// TIA Portal project "Project1" (V14)

(* hardware
DEVICE "S71500/ET200MP station_1"  S7-1500 station
   slot 0: "Rail_0"  Rack  6ES7 590-1***0-0AA0
   slot 1: "PLC_1"  CPU 1516-3 PN/DP  6ES7 516-3AN01-0AB0  V2.1
      slot 3: "CPU display_1"  6ES7591-1BA00-0AA0
   slot 2: "DI 16x24VDC SRC BA_1"  DI 16x24VDC SRC BA  6ES7 521-1BH50-0AA0  V2.0
   slot 3: "DI 16/DQ 16x24VDC/0.5A BA_1"  DI 16/DQ 16x24VDC/0.5A BA  6ES7 523-1BL00-0AA0  V1.0
   slot 4: "AI 8xU/R/RTD/TC HF_1"  AI 8xU/R/RTD/TC HF  6ES7 531-7PF00-0AB0  V1.1
   slot 5: "AQ 4xU/I HF_1"  AQ 4xU/I HF  6ES7 532-5ND00-0AB0  V1.1
   slot 6: "AI/AQ 4xU/I/RTD/TC / 2xU/I ST_1"  AI/AQ 4xU/I/RTD/TC / 2xU/I ST  6ES7 534-7QE00-0AB0  V1.0
   slot 7: "DQ 16x24VDC/0.5A BA_1"  DQ 16x24VDC/0.5A BA  6ES7 522-1BH10-0AA0  V1.0
*)

// ===== PLC "PLC_1"  CPU 1516-3 PN/DP =====

VAR_GLOBAL   // PLC tag table "UP_Robot1"
   "robot1_dc" AT %E0.7 : Bool;
   "robot1_fin_p" AT %E1.0 : Bool;
   "robot1_home" AT %E1.1 : Bool;
   "robot1_temp" AT %T1 : Timer;
   "robot1_cargar" AT %A1.2 : Bool;
   "robot1_descargar" AT %A1.3 : Bool;
   "robot1_b_standby" AT %M1.4 : Bool;   // b = bit
   "robot1_b_ocupacion" AT %M1.5 : Bool;
   "robot1_bdt_carga" AT %M1.6 : Bool;   // bdt = bit de tiempo
   "robot1_bdt_descarga" AT %M1.7 : Bool;
   "robot1_bdc_carga" AT %M2.0 : Bool;   // bdc = bit de configuración
   "robot1_bdc_descarga" AT %M2.1 : Bool;
   "robot1_b_emer" AT %M2.2 : Bool;
   "robot1_emer" AT %M5.7 : Bool;
   "robot1_rearme" AT %M6.0 : Bool;
   "robot1_x_emer" AT %M5.5 : Bool;
   "robot1_x_marcha" AT %M5.6 : Bool;
END_VAR

VAR_GLOBAL   // PLC tag table "UP_Robot2"
   "robot2_dc" AT %E2.5 : Bool;
   "robot2_fin_p" AT %E2.6 : Bool;
   "robot2_home" AT %E3.6 : Bool;
   "robot2_temp" AT %T5 : Timer;
   "robot2_cargar" AT %A6.0 : Bool;
   "robot2_descargar" AT %A6.1 : Bool;
   "robot2_b_standby" AT %M6.2 : Bool;   // b = bit
   "robot2_b_ocupacion" AT %M6.3 : Bool;
   "robot2_bdt_carga" AT %M6.4 : Bool;   // bdt = bit de tiempo
   "robot2_bdt_descarga" AT %M6.5 : Bool;
   "robot2_bdc_carga" AT %M6.6 : Bool;   // bdc = bit de configuración
   "robot2_bdc_descarga" AT %M6.7 : Bool;
   "robot2_b_emer" AT %M7.0 : Bool;
   "robot2_emer" AT %E4.6 : Bool;
   "robot2_rearme" AT %E4.7 : Bool;
END_VAR

VAR_GLOBAL   // PLC tag table "GMM"
   "gmm_on" AT %E0.0 : Bool;
   "gmm_lote_pequenio" AT %E0.1 : Bool;
   "gmm_lote_mediano" AT %E0.2 : Bool;
   "gmm_lote_grande" AT %E0.3 : Bool;
   "gmm_mcong" AT %E0.4 : Bool;
   "gmm_cong" AT %E0.5 : Bool;
   "gmm_bit_marcha" AT %M0.6 : Bool;
   "gmm_bit_paro" AT %M0.7 : Bool;
   "gmm_bit_congelacion" AT %M1.0 : Bool;
END_VAR

VAR_GLOBAL   // PLC tag table "CeldaMecanizado"
   "start" AT %E0.6 : Bool;
END_VAR

VAR_GLOBAL   // PLC tag table "UP_CNC1"
   "cnc1_lapiz" AT %E1.2 : Bool;
   "cnc1_sacapuntas" AT %E1.3 : Bool;
   "cnc1_escuadra" AT %E1.4 : Bool;
   "cnc1_cartabon" AT %E1.5 : Bool;
   "cnc1_home" AT %E1.6 : Bool;
   "cnc1_temp" AT %T2 : Timer;
   "cnc1_cnc_lapiz" AT %A1.7 : Bool;
   "cnc1_cnc_sacapuntas" AT %A2.0 : Bool;
   "cnc1_cnc_escuadra" AT %A2.1 : Bool;
   "cnc1_cnc_cartabon" AT %A2.2 : Bool;
   "cnc1_b_standby" AT %M2.3 : Bool;   // b = bit
   "cnc1_b_ocupacion" AT %M2.4 : Bool;
   "cnc1_bdt_lapiz" AT %M2.5 : Bool;   // bdt = bit de tiempo
   "cnc1_bdt_sacapuntas" AT %M2.6 : Bool;
   "cnc1_bdt_escuadra" AT %M2.7 : Bool;
   "cnc1_bdt_cartabon" AT %M3.0 : Bool;
   "cnc1_bdc_lapiz" AT %M3.1 : Bool;   // bdc = bit de configuración
   "cnc1_bdc_sacapuntas" AT %M3.2 : Bool;
   "cnc1_bdc_escuadra" AT %M3.3 : Bool;
   "cnc1_bdc_cartabon" AT %M3.4 : Bool;
   "cnc1_b_emer" AT %M3.5 : Bool;
   "cnc1_emer" AT %M6.1 : Bool;
   "cnc1_rearme" AT %M7.3 : Bool;
END_VAR

VAR_GLOBAL   // PLC tag table "UP_Simple_Efecto1"
   "sef1_scomp" AT %E1.7 : Bool;   // sef = simple efecto
   "sef1_sexp" AT %E2.0 : Bool;
   "sef1_push" AT %E2.1 : Bool;
   "sef1_temp" AT %T3 : Timer;
   "sef1_expandir" AT %A2.3 : Bool;
   "sef1_b_standby" AT %M3.6 : Bool;   // b = bit
   "sef1_b_ocupacion" AT %M3.7 : Bool;
   "sef1_bdt_expansion" AT %M4.0 : Bool;   // bdt = bit de tiempo
   "sef1_bdt_compresion" AT %M4.1 : Bool;
   "sef1_bdc_expansion" AT %M4.2 : Bool;   // bdc = bit de configuración
   "sef1_bdc_compresion" AT %M4.3 : Bool;
   "sef1_b_emer" AT %M4.4 : Bool;
   "sef1_emer" AT %M9.1 : Bool;
   "sef1_rearme" AT %M9.2 : Bool;
END_VAR

VAR_GLOBAL   // PLC tag table "UT"
   "ut_x0" AT %M4.5 : Bool;
   "ut_m1" AT %M4.6 : Bool;
   "ut_x2" AT %M4.7 : Bool;
   "ut_x10" AT %M5.0 : Bool;
   "ut_r1" AT %E2.2 : Bool;
   "ut_r2" AT %E2.3 : Bool;
   "ut_rearme" AT %E2.4 : Bool;
   "ut_emer" AT %E2.7 : Bool;
   "ut_cong" AT %E3.0 : Bool;
   "ut_sini" AT %E3.1 : Bool;
   "ut_sfin" AT %E3.2 : Bool;
   "ut_reset" AT %E3.3 : Bool;
   "ut_bdt" AT %M5.1 : Bool;   // bdt = bit de tiempo
   "ut_bdc" AT %M5.2 : Bool;   // bdc = bit de configuración
   "ut_bdf" AT %M5.3 : Bool;   // bdf = bit de fin
   "ut_bdo" AT %M5.4 : Bool;   // bdo = bit de ocupación
   "ut_s1" AT %E3.4 : Bool;
   "ut_s2" AT %E3.5 : Bool;
   "ut_temp" AT %T4 : Timer;
   "ut_actuador1" AT %A3.6 : Bool;
END_VAR

VAR_GLOBAL   // PLC tag table "UP_CNC2"
   "cnc2_lapiz" AT %E3.7 : Bool;
   "cnc2_sacapuntas" AT %E4.0 : Bool;
   "cnc2_escuadra" AT %E4.1 : Bool;
   "cnc2_cartabon" AT %E4.2 : Bool;
   "cnc2_home" AT %E4.3 : Bool;
   "cnc2_temp" AT %T6 : Timer;
   "cnc2_cnc_lapiz" AT %A7.0 : Bool;
   "cnc2_cnc_sacapuntas" AT %A7.1 : Bool;
   "cnc2_cnc_escuadra" AT %A7.2 : Bool;
   "cnc2_cnc_cartabon" AT %A7.3 : Bool;
   "cnc2_b_standby" AT %M7.4 : Bool;   // b = bit
   "cnc2_b_ocupacion" AT %M7.5 : Bool;
   "cnc2_bdt_lapiz" AT %M7.6 : Bool;   // bdt = bit de tiempo
   "cnc2_bdt_sacapuntas" AT %M7.7 : Bool;
   "cnc2_bdt_escuadra" AT %M8.0 : Bool;
   "cnc2_bdt_cartabon" AT %M8.1 : Bool;
   "cnc2_bdc_lapiz" AT %M8.2 : Bool;   // bdc = bit de configuración
   "cnc2_bdc_sacapuntas" AT %M8.3 : Bool;
   "cnc2_bdc_escuadra" AT %M8.4 : Bool;
   "cnc2_bdc_cartabon" AT %M8.5 : Bool;
   "cnc2_b_emer" AT %M8.6 : Bool;
   "cnc2_emer" AT %M8.7 : Bool;
   "cnc2_rearme" AT %M9.0 : Bool;
END_VAR

VAR_GLOBAL   // PLC tag table "GEMER"
   "x_emer" AT %M7.1 : Bool;
   "x_marcha" AT %M7.2 : Bool;
   "emer" AT %E5.0 : Bool;
   "rearme" AT %E5.1 : Bool;
   "emer_local_robot1" AT %E5.2 : Bool;
   "rearme_local_robot1" AT %E5.3 : Bool;
   "emer_local_robot2" AT %E5.4 : Bool;
   "rearme_local_robot2" AT %E5.5 : Bool;
   "emer_local_cnc1" AT %E5.6 : Bool;
   "rearme_local_cnc1" AT %E5.7 : Bool;
   "emer_local_simple_efecto1" AT %E6.0 : Bool;
   "rearme_local_simple_efecto1" AT %E6.1 : Bool;
   "emer_local_cnc2" AT %E6.2 : Bool;
   "rearme_local_cnc2" AT %E6.3 : Bool;
   "emer_local_palets_vacios" AT %E6.4 : Bool;
   "rearme_local_palets_vacios" AT %E6.5 : Bool;
END_VAR

VAR_GLOBAL   // PLC tag table "UP_Palets_Vacios"
   "pa_emer" AT %M9.3 : Bool;
   "pa_rearme" AT %M9.4 : Bool;
   "pa_recoger_pila" AT %A9.5 : Bool;
   "pa_pila_saturada" AT %A9.6 : Bool;
   "pa_error_medida" AT %A9.7 : Bool;
   "pa_h<hmin" AT %A10.0 : Bool;
   "pa_h>hmin" AT %A10.1 : Bool;
   "pa_h>hmax" AT %A10.2 : Bool;
   "pa_hreal" AT %AD10 : Real;
   "pa_hraw" AT %EW14 : Int;
END_VAR

// folder: CNC

DATA_BLOCK "UP_CNC1_DB"   // DB4
{ S7_Optimized_Access := 'TRUE' }
VERSION : 0.1
// stored: InstanceOfName UP_CNC
"UP_CNC"
BEGIN
END_DATA_BLOCK

DATA_BLOCK "UP_CNC2_DB"   // DB18
{ S7_Optimized_Access := 'TRUE' }
VERSION : 0.1
// stored: InstanceOfName UP_CNC
"UP_CNC"
BEGIN
END_DATA_BLOCK

// folder: Cilindro simple efecto

DATA_BLOCK "UP_Simple_Efecto1_DB"   // DB10
{ S7_Optimized_Access := 'TRUE' }
VERSION : 0.1
// stored: InstanceOfName UP_Simple_Efecto
"UP_Simple_Efecto"
BEGIN
END_DATA_BLOCK

// folder: Datos producción

DATA_BLOCK "datosProduccion"   // DB1
{ S7_Optimized_Access := 'TRUE' }
VERSION : 0.1
   VAR
      tmax_simple_efecto : S5Time := s5t#5s;   // Tiempo máximo expansión / compresión
      tmax_carga_descarga : S5Time := s5t#10s;   // Tiempo máximo carga / descarga
      tmax_cnc_lapiz : S5Time := s5t#14s;   // Tiempo máximo cnc
      tmax_cnc_sacapuntas : S5Time := s5t#20s;
      tmax_cnc_escuadra : S5Time := s5t#10s;
      tmax_cnc_cartabon : S5Time := s5t#10s;
      LO_LIM : Real := 0.0;
      HI_LIM : Real := 50.0;
      hmin : Real := 25.0;
      hmax : Real := 30.0;
   END_VAR
BEGIN
END_DATA_BLOCK

DATA_BLOCK "datosLotePequenio"   // DB8
{ S7_Optimized_Access := 'TRUE' }
VERSION : 0.1
   VAR
      tmax_cnc_lapiz : S5Time := s5t#7s;   // Tiempo máximo cnc
      tmax_cnc_sacapuntas : S5Time := s5t#10s;
      tmax_cnc_escuadra : S5Time := s5t#5s;
      tmax_cnc_cartabon : S5Time := s5t#5s;
   END_VAR
BEGIN
END_DATA_BLOCK

DATA_BLOCK "datosLoteMediano"   // DB9
{ S7_Optimized_Access := 'TRUE' }
VERSION : 0.1
   VAR
      tmax_cnc_lapiz : S5Time := s5t#14s;   // Tiempo máximo cnc
      tmax_cnc_sacapuntas : S5Time := s5t#20s;
      tmax_cnc_escuadra : S5Time := s5t#10s;
      tmax_cnc_cartabon : S5Time := s5t#10s;
   END_VAR
BEGIN
END_DATA_BLOCK

DATA_BLOCK "datosLoteGrande"   // DB12
{ S7_Optimized_Access := 'TRUE' }
VERSION : 0.1
   VAR
      tmax_cnc_lapiz : S5Time := s5t#21s;   // Tiempo máximo cnc
      tmax_cnc_sacapuntas : S5Time := s5t#30s;
      tmax_cnc_escuadra : S5Time := s5t#15s;
      tmax_cnc_cartabon : S5Time := s5t#15s;
   END_VAR
BEGIN
END_DATA_BLOCK

// folder: Emergencia

DATA_BLOCK "GEMER_Robot1_DB"   // DB5
{ S7_Optimized_Access := 'TRUE' }
VERSION : 0.1
// stored: InstanceOfName GEMER_Local
"GEMER_Local"
BEGIN
END_DATA_BLOCK

DATA_BLOCK "GEMER_Robot2_DB"   // DB6
{ S7_Optimized_Access := 'TRUE' }
VERSION : 0.1
// stored: InstanceOfName GEMER_Local
"GEMER_Local"
BEGIN
END_DATA_BLOCK

DATA_BLOCK "GEMER_CNC1_DB"   // DB19
{ S7_Optimized_Access := 'TRUE' }
VERSION : 0.1
// stored: InstanceOfName GEMER_Local
"GEMER_Local"
BEGIN
END_DATA_BLOCK

DATA_BLOCK "GEMER_CNC2_DB"   // DB20
{ S7_Optimized_Access := 'TRUE' }
VERSION : 0.1
// stored: InstanceOfName GEMER_Local
"GEMER_Local"
BEGIN
END_DATA_BLOCK

DATA_BLOCK "GEMER_Simple_Efecto1_DB"   // DB21
{ S7_Optimized_Access := 'TRUE' }
VERSION : 0.1
// stored: InstanceOfName GEMER_Local
"GEMER_Local"
BEGIN
END_DATA_BLOCK

DATA_BLOCK "GEMER_Local_Palets_Vacios_DB"   // DB22
{ S7_Optimized_Access := 'TRUE' }
VERSION : 0.1
// stored: InstanceOfName GEMER_Local
"GEMER_Local"
BEGIN
END_DATA_BLOCK

// folder: Modos de marcha

DATA_BLOCK "GMM_DB"   // DB2
{ S7_Optimized_Access := 'TRUE' }
VERSION : 0.1
// stored: InstanceOfName GMM
"GMM"
BEGIN
END_DATA_BLOCK

// folder: Palets vacíos

DATA_BLOCK "UP_Palets_Vacios_DB"   // DB7
{ S7_Optimized_Access := 'TRUE' }
VERSION : 0.1
// stored: InstanceOfName UP_Palets_Vacios
"UP_Palets_Vacios"
BEGIN
END_DATA_BLOCK

// folder: Robots carga / descarga

DATA_BLOCK "UP_Robot1_DB"   // DB3
{ S7_Optimized_Access := 'TRUE' }
VERSION : 0.1
// stored: InstanceOfName UP_Robot
"UP_Robot"
BEGIN
END_DATA_BLOCK

DATA_BLOCK "UP_Robot2_DB"   // DB17
{ S7_Optimized_Access := 'TRUE' }
VERSION : 0.1
// stored: InstanceOfName UP_Robot
"UP_Robot"
BEGIN
END_DATA_BLOCK

// folder: Test unitarios

DATA_BLOCK "UT_SFC_Cilindro_DB"   // DB11
{ S7_Optimized_Access := 'TRUE' }
VERSION : 0.1
// stored: InstanceOfName SFC_Cilindro
"SFC_Cilindro"
BEGIN
END_DATA_BLOCK

DATA_BLOCK "UT_SFC_Programa_DB"   // DB13
{ S7_Optimized_Access := 'TRUE' }
VERSION : 0.1
// stored: InstanceOfName SFC_Programa
"SFC_Programa"
BEGIN
END_DATA_BLOCK

DATA_BLOCK "UT_UP_Simple_Efecto_DB"   // DB14
{ S7_Optimized_Access := 'TRUE' }
VERSION : 0.1
// stored: InstanceOfName UP_Simple_Efecto
"UP_Simple_Efecto"
BEGIN
END_DATA_BLOCK

DATA_BLOCK "UT_UP_CNC_DB"   // DB15
{ S7_Optimized_Access := 'TRUE' }
VERSION : 0.1
// stored: InstanceOfName UP_CNC
"UP_CNC"
BEGIN
END_DATA_BLOCK

DATA_BLOCK "UT_UP_Robot_DB"   // DB16
{ S7_Optimized_Access := 'TRUE' }
VERSION : 0.1
// stored: InstanceOfName UP_Robot
"UP_Robot"
BEGIN
END_DATA_BLOCK

DATA_BLOCK "UT_UP_Palets_Vacios_DB"   // DB23
{ S7_Optimized_Access := 'TRUE' }
VERSION : 0.1
// stored: InstanceOfName UP_Palets_Vacios
"UP_Palets_Vacios"
BEGIN
END_DATA_BLOCK

// folder: (top level)

ORGANIZATION_BLOCK "main"   // OB1, STL, ProgramCycle
TITLE = "Main Program Sweep (Cycle)"
{ S7_Optimized_Access := 'TRUE' }
VERSION : 0.1
// Se encarga de llamar a las unidades productivas, integrando los modos de marcha y las emergencias. Llama a los bloques en el siguiente orden:
// - Emergencia global
// - Emergencias locales
// - Rearmes
// - Modos de marcha
// - Unidades productivas
// Las salidas de los bloques de emergencia y modos de marcha determinarán las entradas “emer”, “rearme”, “cong” y “start” de las unidades productivas.
   VAR_INPUT
      Initial_Call : Bool;   // Initial call of this OB
      Remanence : Bool;   // =True, if remanent data are available
   END_VAR
BEGIN

REGION Network 1: Gemer global
   // Llama a la emergencia global.
         CALL  "GEMER_Global";
END_REGION

REGION Network 2: Gemer robot1
   // Si no hay emergencia global, llama a la emergencia del robot 1.
         AN    "x_emer";

         JCN   _emer_robot1;

         CALL  "GEMER_Local", "GEMER_Robot1_DB"
         ( emer     := "emer_local_robot1",
           rearme   := "rearme_local_robot1",
           bit_emer := "robot1_emer"
         );

   _emer_robot1:NOP   0;
END_REGION

REGION Network 3: Gemer robot2
   // Si no hay emergencia global, llama a la emergencia del robot 2.
         AN    "x_emer";

         JCN   _emer_robot2;

         CALL  "GEMER_Local", "GEMER_Robot2_DB"
         ( emer     := "emer_local_robot2",
           rearme   := "rearme_local_robot2",
           bit_emer := "robot2_emer"
         );

   _emer_robot2:NOP   0;
END_REGION

REGION Network 4: Gemer cnc1
   // Si no hay emergencia global, llama a la emergencia del cnc 1.
         AN    "x_emer";

         JCN   _emer_cnc1;

         CALL  "GEMER_Local", "GEMER_CNC1_DB"
         ( emer     := "emer_local_cnc1",
           rearme   := "rearme_local_cnc1",
           bit_emer := "cnc1_emer"
         );

   _emer_cnc1:NOP   0;
END_REGION

REGION Network 5: Gemer cnc2
   // Si no hay emergencia global, llama a la emergencia del cnc 2.
         AN    "x_emer";

         JCN   _emer_cnc2;

         CALL  "GEMER_Local", "GEMER_CNC2_DB"
         ( emer     := "emer_local_cnc2",
           rearme   := "rearme_local_cnc2",
           bit_emer := "cnc2_emer"
         );

   _emer_cnc2:NOP   0;
END_REGION

REGION Network 6: Gemer simple efecto1
         AN    "x_emer";

         JCN   _emer_simple_efecto1;

         CALL  "GEMER_Local", "GEMER_Simple_Efecto1_DB"
         ( emer     := "emer_local_simple_efecto1",
           rearme   := "rearme_local_simple_efecto1",
           bit_emer := "sef1_emer"
         );

   _emer_simple_efecto1:NOP   0;
END_REGION

REGION Network 7: Gemer palets vacíos
         AN    "x_emer";

         JCN   _palets_vacios1;

         CALL  "GEMER_Local", "GEMER_Local_Palets_Vacios_DB"
         ( emer     := "emer_local_palets_vacios",
           rearme   := "rearme_local_palets_vacios",
           bit_emer := "pa_emer"
         );

   _palets_vacios1:NOP   0;
END_REGION

REGION Network 8: Rearme robot1
         O     "rearme";
         O     "rearme_local_robot1";
         =     "robot1_rearme";
END_REGION

REGION Network 9: Rearme robot2
         O     "rearme";
         O     "rearme_local_robot2";
         =     "robot2_rearme";
END_REGION

REGION Network 10: Rearme cnc1
         O     "rearme";
         O     "rearme_local_cnc1";
         =     "cnc1_rearme";
END_REGION

REGION Network 11: Rearme cnc2
         O     "rearme";
         O     "rearme_local_cnc2";
         =     "cnc2_rearme";
END_REGION

REGION Network 12: Rearme simple efecto1
         O     "rearme";
         O     "rearme_local_simple_efecto1";
         =     "sef1_rearme";
END_REGION

REGION Network 13: Rearme palets vacíos
         O     "rearme";
         O     "rearme_local_palets_vacios";
         =     "pa_rearme";
END_REGION

REGION Network 14: GMM
   // Si no hay emergencia global, se ejecutan los modos de marcha. En caso contrario, se ejecutarán desde GEMER_Global, que activará la plantilla de desconexión:
         AN    "x_emer";

         JCN   _gmm_emer;

         CALL  "GMM", "GMM_DB"
         ( on              := "gmm_on",
           lote_pequenio   := "gmm_lote_pequenio",
           lote_mediano    := "gmm_lote_mediano",
           lote_grande     := "gmm_lote_grande",
           mcong           := "gmm_mcong",
           cong            := "gmm_cong",
           emer            := FALSE,
           bit_paro        := "gmm_bit_paro",
           bit_marcha      := "gmm_bit_marcha",
           bit_congelacion := "gmm_bit_congelacion"
         );

   _gmm_emer:NOP   0;
END_REGION

REGION Network 15: UP_Robot1
         CALL  "UP_Robot", "UP_Robot1_DB"
         ( start                     := "gmm_bit_marcha",
           emer                      := "robot1_emer",
           rearme                    := "robot1_rearme",
           cong                      := "gmm_bit_congelacion",
           dc                        := "robot1_dc",
           fin_p                     := "robot1_fin_p",
           home                      := "robot1_home",
           tiempo_max                := "datosProduccion".tmax_carga_descarga,
           temp_max                  := "robot1_temp",
           cargar                    := "robot1_cargar",
           descargar                 := "robot1_descargar",
           bit_standby               := "robot1_b_standby",
           bit_ocupacion             := "robot1_b_ocupacion",
           bit_error_tiempo_carga    := "robot1_bdt_carga",
           bit_error_tiempo_descarga := "robot1_bdt_descarga",
           bit_error_config_carga    := "robot1_bdc_carga",
           bit_error_config_descarga := "robot1_bdc_descarga",
           bit_emer                  := "robot1_b_emer"
         );
END_REGION

REGION Network 16: UP_Robot2
         CALL  "UP_Robot", "UP_Robot2_DB"
         ( start                     := "gmm_bit_marcha",
           emer                      := "robot2_emer",
           rearme                    := "robot2_rearme",
           cong                      := "gmm_bit_congelacion",
           dc                        := "robot2_dc",
           fin_p                     := "robot2_fin_p",
           home                      := "robot2_home",
           tiempo_max                := "datosProduccion".tmax_carga_descarga,
           temp_max                  := "robot2_temp",
           cargar                    := "robot2_cargar",
           descargar                 := "robot2_descargar",
           bit_standby               := "robot2_b_standby",
           bit_ocupacion             := "robot2_b_ocupacion",
           bit_error_tiempo_carga    := "robot2_bdt_carga",
           bit_error_tiempo_descarga := "robot2_bdt_descarga",
           bit_error_config_carga    := "robot2_bdc_carga",
           bit_error_config_descarga := "robot2_bdc_descarga",
           bit_emer                  := "robot2_b_emer"
         );
END_REGION

REGION Network 17: UP_CNC1
         CALL  "UP_CNC", "UP_CNC1_DB"
         ( start                       := "gmm_bit_marcha",
           emer                        := "cnc1_emer",
           rearme                      := "cnc1_rearme",
           cong                        := "gmm_bit_congelacion",
           lapiz                       := "cnc1_lapiz",
           sacapuntas                  := "cnc1_sacapuntas",
           escuadra                    := "cnc1_escuadra",
           cartabon                    := "cnc1_cartabon",
           home                        := "cnc1_home",
           tmax_cnc_lapiz              := "datosProduccion".tmax_cnc_lapiz,
           tmax_cnc_sacapuntas         := "datosProduccion".tmax_cnc_sacapuntas,
           tmax_cnc_escuadra           := "datosProduccion".tmax_cnc_escuadra,
           tmax_cnc_cartabon           := "datosProduccion".tmax_cnc_cartabon,
           temp_max                    := "cnc1_temp",
           cnc_lapiz                   := "cnc1_cnc_lapiz",
           cnc_sacapuntas              := "cnc1_cnc_sacapuntas",
           cnc_escuadra                := "cnc1_cnc_escuadra",
           cnc_cartabon                := "cnc1_cnc_cartabon",
           bit_standby                 := "cnc1_b_standby",
           bit_ocupacion               := "cnc1_b_ocupacion",
           bit_error_tiempo_lapiz      := "cnc1_bdt_lapiz",
           bit_error_tiempo_sacapuntas := "cnc1_bdt_sacapuntas",
           bit_error_tiempo_escuadra   := "cnc1_bdt_escuadra",
           bit_error_tiempo_cartabon   := "cnc1_bdt_cartabon",
           bit_error_config_lapiz      := "cnc1_bdc_lapiz",
           bit_error_config_sacapuntas := "cnc1_bdc_sacapuntas",
           bit_error_config_escuadra   := "cnc1_bdc_escuadra",
           bit_error_config_cartabon   := "cnc1_bdc_cartabon",
           bit_emer                    := "cnc1_b_emer"
         );
END_REGION

REGION Network 18: UP_CNC2
         CALL  "UP_CNC", "UP_CNC2_DB"
         ( start                       := "gmm_bit_marcha",
           emer                        := "cnc2_emer",
           rearme                      := "cnc2_rearme",
           cong                        := "gmm_bit_congelacion",
           lapiz                       := "cnc2_lapiz",
           sacapuntas                  := "cnc2_sacapuntas",
           escuadra                    := "cnc2_escuadra",
           cartabon                    := "cnc2_cartabon",
           home                        := "cnc2_home",
           tmax_cnc_lapiz              := "datosProduccion".tmax_cnc_lapiz,
           tmax_cnc_sacapuntas         := "datosProduccion".tmax_cnc_sacapuntas,
           tmax_cnc_escuadra           := "datosProduccion".tmax_cnc_escuadra,
           tmax_cnc_cartabon           := "datosProduccion".tmax_cnc_cartabon,
           temp_max                    := "cnc2_temp",
           cnc_lapiz                   := "cnc2_cnc_lapiz",
           cnc_sacapuntas              := "cnc2_cnc_sacapuntas",
           cnc_escuadra                := "cnc2_cnc_escuadra",
           cnc_cartabon                := "cnc2_cnc_cartabon",
           bit_standby                 := "cnc2_b_standby",
           bit_ocupacion               := "cnc2_b_ocupacion",
           bit_error_tiempo_lapiz      := "cnc2_bdt_lapiz",
           bit_error_tiempo_sacapuntas := "cnc2_bdt_sacapuntas",
           bit_error_tiempo_escuadra   := "cnc2_bdt_escuadra",
           bit_error_tiempo_cartabon   := "cnc2_bdt_cartabon",
           bit_error_config_lapiz      := "cnc2_bdc_lapiz",
           bit_error_config_sacapuntas := "cnc2_bdc_sacapuntas",
           bit_error_config_escuadra   := "cnc2_bdc_escuadra",
           bit_error_config_cartabon   := "cnc2_bdc_cartabon",
           bit_emer                    := "cnc2_b_emer"
         );
END_REGION

REGION Network 19: UP_Simple_Efecto1
         CALL  "UP_Simple_Efecto", "UP_Simple_Efecto1_DB"
         ( start                       := "gmm_bit_marcha",
           emer                        := "sef1_emer",
           cong                        := "sef1_rearme",
           rearme                      := "gmm_bit_congelacion",
           scomp                       := "sef1_scomp",
           sexp                        := "sef1_sexp",
           push                        := "sef1_push",
           tiempo_max                  := "datosProduccion".tmax_simple_efecto,
           temp_max                    := "sef1_temp",
           expandir                    := "sef1_expandir",
           bit_standby                 := "sef1_b_standby",
           bit_ocupacion               := "sef1_b_ocupacion",
           bit_error_tiempo_expansion  := "sef1_bdt_expansion",
           bit_error_tiempo_compresion := "sef1_bdt_compresion",
           bit_error_config_expansion  := "sef1_bdc_expansion",
           bit_error_config_compresion := "sef1_bdc_expansion",
           bit_emer                    := "sef1_b_emer"
         );
END_REGION

REGION Network 20: UP_Palets_Vacios
         CALL  "UP_Palets_Vacios","UP_Palets_Vacios_DB"
         ( start         := "gmm_bit_marcha",
           emer          := "pa_emer",
           rearme        := "pa_rearme",
           cong          := "gmm_bit_congelacion",
           hraw          := "pa_hraw",
           LO_LIM        := "datosProduccion".LO_LIM,
           HI_LIM        := "datosProduccion".HI_LIM,
           hmin          := "datosProduccion".hmin,
           hmax          := "datosProduccion".hmax,
           recoger_pila  := "pa_recoger_pila",
           pila_saturada := "pa_pila_saturada",
           error_medida  := "pa_error_medida",
           h_real        := "pa_hreal",
           "h>hmin"      := "pa_h>hmin",
           "h>hmax"      := "pa_h>hmax",
           "h<hmin"      := "pa_h<hmin"
         );
END_REGION
END_ORGANIZATION_BLOCK

ORGANIZATION_BLOCK "init"   // OB100, STL, Startup
TITLE = "Complete Restart"
{ S7_Optimized_Access := 'TRUE' }
VERSION : 0.1
   VAR_INPUT
      LostRetentive : Bool;   // True if retentive data are lost
      LostRTC : Bool;   // True if date and time are lost
   END_VAR
BEGIN

REGION Network 1: Inicialización
         SET;
         S     "x_marcha";
         R     "x_emer";
END_REGION
END_ORGANIZATION_BLOCK

// folder: CNC

FUNCTION_BLOCK "UP_CNC"   // FB8, STL
TITLE = Unidad productiva CNC
{ S7_Optimized_Access := 'TRUE' }
VERSION : 0.1
// Gestiona la CNC.
// Presenta los siguientes parámetros:
// - start: inicia la unidad productiva.
// - emer: señal de emergencia (error asíncrono).
// - cong: señal de congelación.
// - rearme: vuelta al estado de standby de un estado de error.
// - lapiz: indica que se van a procesar lápices.
// - sacapuntas: indica que se van a procesar sacapuntas.
// - escuadra: indica que se van a procesar escuadras.
// - cartabon: indica que se van a procesar cartabones.
// - home: indica el estado en la posición fetal.
// - tmax_cnc_lapiz: tiempo máximo para la fabricación del lápiz.
// - tmax_cnc_sacapuntas: tiempo máximo para la fabricación del sacapuntas.
// - tmax_cnc_escuadra: tiempo máximo para la fabricación de la escuadra.
// - tmax_cnc_cartabon: tiempo máximo para la fabricación del cartabón.
// - temp_max: temporizador de las manioabras.
// - cnc_lapiz: programa del lápiz.
// - cnc_sacapuntas: programa del sacapuntas.
// - cnc_escuadra: programa de la escuadra.
// - cnc_cartabon: programa del cartabón.
// - bit_standby: estado de standby.
// - bit_ocupación: el robot se encuentra en medio de una maniobra.
// - bit_error_tiempo_lapiz: error síncrono en la lápiz.
// - bit_error_tiempo_sacapuntas: error síncrono en la sacapuntas.
// - bit_error_tiempo_escuadra: error síncrono en las escuadras.
// - bit_error_tiempo_cartabon: error síncrono en los cartabones.
// - bit_error_config_lapiz: error síncrono por mala configuración inicial en la fabricación del lápiz.
// - bit_error_config_sacapuntas: error síncrono por mala configuración inicial en la fabricación del sacapuntas.
// - bit_error_config_escuadras: error síncrono por mala configuración inicial en la fabricación de la escuadra.
// - bit_error_config_cartabon: error síncrono por mala configuración inicial en la fabricación del cartabón.
// - bit_emer: estado de emergencia.
// - bit_trabajo: se encarga de la conexión de la unidad productiva.
// - x_carga: estado de carga.
// - x_descarga: estado de descarga.
// - x_standby: estado de standby.
// - x_error_tiempo_lapiz: estado de error síncrono en la fabricación del lápiz.
// - x_error_tiempo_sacapuntas: estado de error síncrono en la la fabricación del sacapuntas.
// - x_error_tiempo_escuadra: estado de error síncrono en la fabricación de la escuadra.
// - x_error_tiempo_cartabon: estado de error síncrono en la la fabricación del cartabón.
// - x_error_config_lapiz: estado de error síncrono por mala configuración inicial en la fabricación del lápiz.
// - x_error_config_sacapuntas: estado de error síncrono por mala configuración inicial en la fabricación del sacapuntas.
// - x_error_config_escuadra: estado de error síncrono por mala configuración inicial en la fabricación del lápiz.
// - x_error_config_cartabon: estado de error síncrono por mala configuración inicial en la fabricación del cartabon.
// - x_emer: estado de emergencia por error asíncrono.
// - SFC_lapiz: maniobra para la fabricación del lápiz de tipo SFC_Programa con bloque de datos multiinstancia.
// - SFC_sacapuntas:  maniobra para la fabricación del sacapuntas de tipo SFC_Programa con bloque de datos multiinstancia.
// - SFC_escuadra:  maniobra para la fabricación de la escuadra de tipo SFC_Programa con bloque de datos multiinstancia.
// - SFC_cartabon:  maniobra para la fabricación del cartabon de tipo SFC_Programa con bloque de datos multiinstancia.
// - bit_fin_lápiz: finalización de la fabricación del lápiz.
// - bit_fin_sacapuntas: finalización de la fabricación del sacapuntas. 
// - bit_fin_escuadra: finalización de la fabricación de la escuadra.
// - bit_fin_cartabón: finalización de la fabricación del cartabón. 
// 
// 
// Los bits de fin son temporales porque las unidades productivas están pensadas para estar trabajando constantemente.
   VAR_INPUT
      start : Bool;
      emer : Bool;
      rearme : Bool;
      cong : Bool;
      lapiz : Bool;
      sacapuntas : Bool;
      escuadra : Bool;
      cartabon : Bool;
      home : Bool;
      tmax_cnc_lapiz : S5Time;
      tmax_cnc_sacapuntas : S5Time;
      tmax_cnc_escuadra : S5Time;
      tmax_cnc_cartabon : S5Time;
      temp_max : Timer;
   END_VAR
   VAR_OUTPUT
      cnc_lapiz : Bool;
      cnc_sacapuntas : Bool;
      cnc_escuadra : Bool;
      cnc_cartabon : Bool;
      bit_standby : Bool;
      bit_ocupacion : Bool;
      bit_error_tiempo_lapiz : Bool;
      bit_error_tiempo_sacapuntas : Bool;
      bit_error_tiempo_escuadra : Bool;
      bit_error_tiempo_cartabon : Bool;
      bit_error_config_lapiz : Bool;
      bit_error_config_sacapuntas : Bool;
      bit_error_config_escuadra : Bool;
      bit_error_config_cartabon : Bool;
      bit_emer : Bool;
   END_VAR
   VAR
      bit_trabajo : Bool;
      x_lapiz : Bool;
      x_sacapuntas : Bool;
      x_escuadra : Bool;
      x_cartabon : Bool;
      x_standby : Bool;
      x_error_tiempo_lapiz : Bool;
      x_error_tiempo_sacapuntas : Bool;
      x_error_tiempo_escuadra : Bool;
      x_error_tiempo_cartabon : Bool;
      x_error_config_lapiz : Bool;
      x_error_config_sacapuntas : Bool;
      x_error_config_escuadra : Bool;
      x_error_config_cartabon : Bool;
      x_emer : Bool;
      SFC_lapiz : "SFC_Programa";
      SFC_sacapuntas : "SFC_Programa";
      SFC_Escuadra : "SFC_Programa";
      SFC_Cartabon : "SFC_Programa";
   END_VAR
   VAR_TEMP
      bit_fin_lapiz : Bool;
      bit_fin_sacapuntas : Bool;
      bit_fin_escuadra : Bool;
      bit_fin_cartabon : Bool;
   END_VAR
BEGIN

REGION Network 1: Plantilla de desconexión - Error asíncrono
   // Si se está en un estado de error síncrono no se entra en emergencia.
         O     #x_standby;
         O     #x_lapiz;
         O     #x_sacapuntas;
         O     #x_cartabon;
         O     #x_escuadra;
         A     #emer;
         S     #x_emer;
         R     #x_standby;
         R     #x_lapiz;
         R     #x_sacapuntas;
         R     #x_cartabon;
         R     #x_escuadra;

         JCN   _emer;

         CALL  #SFC_lapiz
         ( sensor1          := ,
           sensor2          := ,
           reset            := true,
           tiempo_error     := ,
           temp_error       := ,
           bit_fin          := ,
           bit_error_tiempo := ,
           bit_error_config := ,
           bit_ocupacion    := ,
           actuador1        := #cnc_lapiz
         );

         CALL  #SFC_sacapuntas
         ( sensor1          := ,
           sensor2          := ,
           reset            := true,
           tiempo_error     := ,
           temp_error       := ,
           bit_fin          := ,
           bit_error_tiempo := ,
           bit_error_config := ,
           bit_ocupacion    := ,
           actuador1        := #cnc_sacapuntas
         );

         CALL  #SFC_Escuadra
         ( sensor1          := ,
           sensor2          := ,
           reset            := TRUE,
           tiempo_error     := ,
           temp_error       := ,
           bit_fin          := ,
           bit_error_tiempo := ,
           bit_error_config := ,
           bit_ocupacion    := ,
           actuador1        := #cnc_escuadra
         );

         CALL  #SFC_Cartabon
         ( sensor1          := ,
           sensor2          := ,
           reset            := TRUE,
           tiempo_error     := ,
           temp_error       := ,
           bit_fin          := ,
           bit_error_tiempo := ,
           bit_error_config := ,
           bit_ocupacion    := ,
           actuador1        := #cnc_cartabon
         );

   _emer:NOP   0;

         O     #x_standby;
         O     #x_lapiz;
         O     #x_sacapuntas;
         O     #x_cartabon;
         O     #x_escuadra;
         A     #emer;
         BEC;
END_REGION

REGION Network 2: Plantilla de desconexión - STOP
   // Desconexión de la unidad productiva. 
   // Reinicia todos los parámetros para futuras conexiones.
   // Llamada a las maniobras usando la entrada asíncrona para indicar su pausa.
   // Después de la caja de código se especifica la instrucción “UN #start”, que coincide con la instrucción con la que se activó la plantilla. Esto es porque después de la caja, la RLO = 1 y /ER = 0. Por lo tanto, si la plantilla no se ejecuta, tras saltar la caja de código la RLO = 1 cuando debería ser 0 (UN #start no se cumple).
         AN    #start;
         R     #bit_trabajo;
         R     #bit_emer;
         R     #bit_error_config_lapiz;
         R     #bit_error_config_sacapuntas;
         R     #bit_error_tiempo_lapiz;
         R     #bit_error_tiempo_sacapuntas;
         R     #bit_standby;
         R     #bit_ocupacion;
         R     #temp_max;
         FR    #temp_max;

         JCN   stop;

         CALL  #SFC_lapiz
         ( sensor1          := ,
           sensor2          := ,
           reset            := true,
           tiempo_error     := ,
           temp_error       := ,
           bit_fin          := ,
           bit_error_tiempo := ,
           bit_error_config := ,
           bit_ocupacion    := ,
           actuador1        := #cnc_lapiz
         );

         CALL  #SFC_sacapuntas
         ( sensor1          := ,
           sensor2          := ,
           reset            := true,
           tiempo_error     := ,
           temp_error       := ,
           bit_fin          := ,
           bit_error_tiempo := ,
           bit_error_config := ,
           bit_ocupacion    := ,
           actuador1        := #cnc_sacapuntas
         );

         CALL  #SFC_Escuadra
         ( sensor1          := ,
           sensor2          := ,
           reset            := TRUE,
           tiempo_error     := ,
           temp_error       := ,
           bit_fin          := ,
           bit_error_tiempo := ,
           bit_error_config := ,
           bit_ocupacion    := ,
           actuador1        := #cnc_sacapuntas
         );

         CALL  #SFC_Cartabon
         ( sensor1          := ,
           sensor2          := ,
           reset            := TRUE,
           tiempo_error     := ,
           temp_error       := ,
           bit_fin          := ,
           bit_error_tiempo := ,
           bit_error_config := ,
           bit_ocupacion    := ,
           actuador1        := #cnc_cartabon
         );

   stop: NOP   0;

         AN    #start;
         BEC;
END_REGION

REGION Network 3: Plantilla de conexión
   // Conexión de la unidad productiva.
         A     #start;
         FP    #bit_trabajo;
         S     #x_standby;
         R     #x_lapiz;
         R     #x_sacapuntas;
         R     #x_cartabon;
         R     #x_escuadra;
         R     #x_emer;
         R     #x_error_config_lapiz;
         R     #x_error_config_sacapuntas;
         R     #x_error_config_escuadra;
         R     #x_error_config_cartabon;
         R     #x_error_tiempo_lapiz;
         R     #x_error_tiempo_sacapuntas;
         R     #x_error_tiempo_escuadra;
         R     #x_error_tiempo_cartabon;
END_REGION

REGION Network 4: Plantilla de congelación
   // Congela la unidad productiva: habilita los componentes y resetea los actuadores (llamadas a maniobras).
   // Se repite el estimulo de activación de la plantilla antes de la instrucción "BEB" para asegurar la salida del bloque.
         A     #cong;

         JCN   _cong;

         R     #temp_max;  //Habilitación de componentes
         FR    #temp_max;

         CALL  #SFC_lapiz
         ( sensor1          := ,
           sensor2          := ,
           reset            := TRUE,
           tiempo_error     := ,
           temp_error       := ,
           bit_fin          := ,
           bit_error_tiempo := ,
           bit_error_config := ,
           bit_ocupacion    := ,
           actuador1        := #cnc_lapiz
         );

         CALL  #SFC_sacapuntas
         ( sensor1          := ,
           sensor2          := ,
           reset            := TRUE,
           tiempo_error     := ,
           temp_error       := ,
           bit_fin          := ,
           bit_error_tiempo := ,
           bit_error_config := ,
           bit_ocupacion    := ,
           actuador1        := #cnc_sacapuntas
         );

         CALL  #SFC_Escuadra
         ( sensor1          := ,
           sensor2          := ,
           reset            := TRUE,
           tiempo_error     := ,
           temp_error       := ,
           bit_fin          := ,
           bit_error_tiempo := ,
           bit_error_config := ,
           bit_ocupacion    := ,
           actuador1        := #cnc_escuadra
         );

         CALL  #SFC_Cartabon
         ( sensor1          := ,
           sensor2          := ,
           reset            := TRUE,
           tiempo_error     := ,
           temp_error       := ,
           bit_fin          := ,
           bit_error_tiempo := ,
           bit_error_config := ,
           bit_ocupacion    := ,
           actuador1        := #cnc_cartabon
         );

   _cong:NOP   0;

         A     #cong;  //Repetición del estímulo de activación
         BEC;
END_REGION

REGION Network 5: Salida del estado de emergencia
   // Rearme
         A     #x_emer;
         AN    #emer;
         A     #rearme;
         S     #x_standby;
         R     #x_emer;
END_REGION

REGION Network 6: Rearme errores síncronos
   // Se considera la posibilidad de rearme tras errores síncronos.
         O     #x_error_config_lapiz;
         O     #x_error_config_sacapuntas;
         O     #x_error_config_escuadra;
         O     #x_error_config_cartabon;
         O     #x_error_tiempo_lapiz;
         O     #x_error_tiempo_sacapuntas;
         O     #x_error_tiempo_escuadra;
         O     #x_error_tiempo_cartabon;
         A     #rearme;
         S     #x_standby;
         R     #x_error_config_lapiz;
         R     #x_error_config_sacapuntas;
         R     #x_error_config_escuadra;
         R     #x_error_config_cartabon;
         R     #x_error_tiempo_lapiz;
         R     #x_error_tiempo_sacapuntas;
         R     #x_error_tiempo_escuadra;
         R     #x_error_tiempo_cartabon;
END_REGION

REGION Network 7: x_standby -> x_lapiz
         A     #x_standby;
         A     #lapiz;
         S     #x_lapiz;
         R     #x_standby;
END_REGION

REGION Network 8: x_standby -> x_sacapuntas
         A     #x_standby;
         A     #sacapuntas;
         S     #x_sacapuntas;
         R     #x_standby;
END_REGION

REGION Network 9: x_standby -> x_escuadra
         A     #x_standby;
         A     #escuadra;
         S     #x_escuadra;
         R     #x_standby;
END_REGION

REGION Network 10: x_standby -> x_cartabon
         A     #x_standby;
         A     #cartabon;
         S     #x_cartabon;
         R     #x_standby;
END_REGION

REGION Network 11: Llamada a la maniobra de fabricación del lápiz
   // Entrada de error asíncrono false (se gestiona en la plantilla de desconexión).
         A     #x_lapiz;

         JCN   _lapiz;
         CALL  #SFC_lapiz
         ( sensor1          := #lapiz,
           sensor2          := #home,
           reset            := false,
           tiempo_error     := #tmax_cnc_lapiz,
           temp_error       := #temp_max,
           bit_fin          := #bit_fin_lapiz,
           bit_error_tiempo := #bit_error_tiempo_lapiz,
           bit_error_config := #bit_error_config_lapiz,
           bit_ocupacion    := #bit_ocupacion,
           actuador1        := #cnc_lapiz
         );

         A     #bit_error_tiempo_lapiz;
         S     #x_error_tiempo_lapiz;
         R     #x_lapiz;

         A     #bit_error_config_lapiz;
         S     #x_error_config_lapiz;
         R     #x_lapiz;

         A     #bit_fin_lapiz;
         S     #x_standby;
         R     #x_lapiz;

   _lapiz:NOP   0;
END_REGION

REGION Network 12: Llamada a la maniobra de fabricación del sacapuntas
         A     #x_sacapuntas;

         JCN   _sacapuntas;
         CALL  #SFC_sacapuntas
         ( sensor1          := #sacapuntas,
           sensor2          := #home,
           reset            := false,
           tiempo_error     := #tmax_cnc_sacapuntas,
           temp_error       := #temp_max,
           bit_fin          := #bit_fin_sacapuntas,
           bit_error_tiempo := #bit_error_tiempo_sacapuntas,
           bit_error_config := #bit_error_config_sacapuntas,
           bit_ocupacion    := #bit_ocupacion,
           actuador1        := #cnc_sacapuntas
         );


         A     #bit_error_tiempo_sacapuntas;
         S     #x_error_tiempo_sacapuntas;
         R     #x_sacapuntas;

         A     #bit_error_config_sacapuntas;
         S     #x_error_config_sacapuntas;
         R     #x_sacapuntas;

         A     #bit_fin_sacapuntas;
         S     #x_standby;
         R     #x_sacapuntas;

   _sacapuntas:NOP   0;
END_REGION

REGION Network 13: Llamada a la maniobra de fabricación del sacapuntas
         A     #x_escuadra;

         JCN   _escuadra;
         CALL  #SFC_Escuadra
         ( sensor1          := #escuadra,
           sensor2          := #home,
           reset            := false,
           tiempo_error     := #tmax_cnc_escuadra,
           temp_error       := #temp_max,
           bit_fin          := #bit_fin_escuadra,
           bit_error_tiempo := #bit_error_tiempo_escuadra,
           bit_error_config := #bit_error_config_escuadra,
           bit_ocupacion    := #bit_ocupacion,
           actuador1        := #cnc_escuadra
         );


         A     #bit_error_tiempo_escuadra;
         S     #x_error_tiempo_escuadra;
         R     #x_escuadra;

         A     #bit_error_config_escuadra;
         S     #x_error_config_escuadra;
         R     #x_escuadra;

         A     #bit_fin_escuadra;
         S     #x_standby;
         R     #x_escuadra;

   _escuadra:NOP   0;
END_REGION

REGION Network 14: Llamada a la maniobra de fabricación del sacapuntas
         A     #x_cartabon;

         JCN   _cartabon;
         CALL  #SFC_Cartabon
         ( sensor1          := #cartabon,
           sensor2          := #home,
           reset            := false,
           tiempo_error     := #tmax_cnc_cartabon,
           temp_error       := #temp_max,
           bit_fin          := #bit_fin_cartabon,
           bit_error_tiempo := #bit_error_tiempo_cartabon,
           bit_error_config := #bit_error_config_cartabon,
           bit_ocupacion    := #bit_ocupacion,
           actuador1        := #cnc_cartabon
         );


         A     #bit_error_tiempo_cartabon;
         S     #x_error_tiempo_cartabon;
         R     #x_cartabon;

         A     #bit_error_config_cartabon;
         S     #x_error_config_cartabon;
         R     #x_cartabon;

         A     #bit_fin_cartabon;
         S     #x_standby;
         R     #x_cartabon;

   _cartabon:NOP   0;
END_REGION

REGION Network 15: Bit de standby
   // Indica el estado de standby.
         A     #x_standby;
         =     #bit_standby;
END_REGION

REGION Network 16: Bit de emergencia
   // Indica el estado de emergencia.
         A     #x_emer;
         =     #bit_emer;
END_REGION

REGION Network 17: Bit error tiempo lápiz
   // Indica el estado de error síncrono por tiempo de fabricación del lápiz.
         A     #x_error_tiempo_lapiz;
         =     #bit_error_tiempo_lapiz;
END_REGION

REGION Network 18: Bit error tiempo sacapuntas
   // Indica el estado de error síncrono por tiempo de fabricación del sacapuntas.
         A     #x_error_tiempo_sacapuntas;
         =     #bit_error_tiempo_sacapuntas;
END_REGION

REGION Network 19: Bit error tiempo escuadra
   // Indica el estado de error síncrono por tiempo de fabricación de la escuadra.
         A     #x_error_tiempo_escuadra;
         =     #bit_error_tiempo_escuadra;
END_REGION

REGION Network 20: Bit error tiempo cartabón
   // Indica el estado de error síncrono por tiempo de fabricación del cartabón.
         A     #x_error_tiempo_cartabon;
         =     #bit_error_tiempo_cartabon;
END_REGION

REGION Network 21: Bit error config lápiz
   // Indica el estado de error síncrono por mala configuración inicial en la fabricación del lápiz.
         A     #x_error_config_lapiz;
         =     #bit_error_config_lapiz;
END_REGION

REGION Network 22: Bit error config sacapuntas
   // Indica el estado de error síncrono por mala configuración inicial en la fabricación del sacapuntas.
         A     #x_error_config_sacapuntas;
         =     #bit_error_config_sacapuntas;
END_REGION

REGION Network 23: Bit error config escuadra
   // Indica el estado de error síncrono por mala configuración inicial en la fabricación de la escuadra.
         A     #x_error_config_escuadra;
         =     #bit_error_config_escuadra;
END_REGION

REGION Network 24: Bit error config cartabón
   // Indica el estado de error síncrono por mala configuración inicial en la fabricación del cartabón.
         A     #x_error_config_cartabon;
         =     #bit_error_config_cartabon;
END_REGION
END_FUNCTION_BLOCK

// folder: Cilindro simple efecto

FUNCTION_BLOCK "UP_Simple_Efecto"   // FB9, STL
TITLE = Unidad productiva cilindro de simple efecto
{ S7_Optimized_Access := 'TRUE' }
VERSION : 0.1
// Gestiona el cilindro de simple efecto.
// Presenta los siguientes parámetros:
// - start: inicia la unidad productiva.
// - emer: señal de emergencia (error asíncrono).
// - cong: señal de congelación. 
// - rearme: vuelta al estado de standby de un estado de error.
// - scomp: cilindro comprimido.
// - sexp: cilindro expandido.
// - push: autorización para expandirse.
// - tiempo_max: tiempo máximo para las maniobras.
// - temp_max: temporizador de las manioabras.
// - expandir: expande el cilindro (no hace falta actuador para comprimir porque es un simple efecto).
// - bit_standby: estado de standby.
// - bit_ocupación: el robot se encuentra en medio de una maniobra.
// - bit_error_tiempo_expansión: error síncrono en la expansión.
// - bit_error_tiempo_compresión: error síncrono en la compresión.
// - bit_error_config_expansión: error síncrono por mala configuración inicial en la expansión.
// - bit_error_config_compresión: error síncrono por mala configuración inicial en la compresión.
// - bit_emer: estado de emergencia.
// - bit_trabajo: se encarga de la conexión de la unidad productiva.
// - x_expansión: estado de expansión.
// - x_compresión: estado de compresión.
// - x_standby: estado de standby.
// - x_error_tiempo_expansión: estado de error síncrono en la expansión.
// - x_error_tiempo_compresión: estado de error síncrono en la compresión.
// - x_error_config_expansión: estado de error síncrono por mala configuración inicial en la expansión.
// - x_error_config_compresión: estado de error síncrono por mala configuración inicial en la compresión.
// - x_emer: estado de error asíncrono.
// - SFC_Expansion: maniobra de expansión.
// - SFC_Compresión: maniobra de compresión (sin actuador).
// - bit_fin_expansión: finalización de la expansión.
// - bit_fin_compresión: finalización de la compresión. 
// 
// 
// No se tiene un actuador "compresion" porque el cilindro es un simple efecto. No actuar sobre el cilindro supone la compresión. Si se definiese un estado de compresión, habría conflictos porque al entrar en emergencia, se llamaría al mismo actuador con "expansion" = 1 y "compresion" = 1.
// Sin embargo, es necesario llamar a la maniobra de compresión para encapsularla y gestionar errores por tiempo y mala configuración inicial.
   VAR_INPUT
      start : Bool;
      emer : Bool;
      cong : Bool;
      rearme : Bool;
      scomp : Bool;
      sexp : Bool;
      push : Bool;
      tiempo_max : S5Time;
      temp_max : Timer;
   END_VAR
   VAR_OUTPUT
      expandir : Bool;
      bit_standby : Bool;
      bit_ocupacion : Bool;
      bit_error_tiempo_expansion : Bool;
      bit_error_tiempo_compresion : Bool;
      bit_error_config_expansion : Bool;
      bit_error_config_compresion : Bool;
      bit_emer : Bool;
   END_VAR
   VAR
      bit_trabajo : Bool;
      x_expansion : Bool;
      x_compresion : Bool;
      x_standby : Bool;
      x_error_tiempo_expansion : Bool;
      x_error_tiempo_compresion : Bool;
      x_error_config_expansion : Bool;
      x_error_config_compresion : Bool;
      x_emer : Bool;
      SFC_Expansion : "SFC_Cilindro";
      SFC_Compresion : "SFC_Cilindro";
   END_VAR
   VAR_TEMP
      bit_fin_expansion : Bool;
      bit_fin_compresion : Bool;
   END_VAR
BEGIN

REGION Network 1: Plantilla de emergencia - Error asíncrono
   // Si se está en un estado de error síncrono no se entra en emergencia.
         O     #x_standby;
         O     #x_expansion;
         O     #x_compresion;
         A     #emer;
         S     #x_emer;
         R     #x_standby;
         R     #x_compresion;
         R     #x_expansion;

         JCN   _emer;

         CALL  #SFC_Expansion
         ( sini             := ,
           sfin             := ,
           reset            := TRUE,
           tiempo_error     := ,
           temp_error       := ,
           bit_fin          := ,
           bit_error_tiempo := ,
           bit_error_config := ,
           bit_ocupacion    := ,
           actuador         := #expandir
         );


         CALL  #SFC_Compresion
         ( sini             := ,
           sfin             := ,
           reset            := TRUE,
           tiempo_error     := ,
           temp_error       := ,
           bit_fin          := ,
           bit_error_tiempo := ,
           bit_error_config := ,
           bit_ocupacion    := ,
           actuador         :=
         );

   _emer:NOP   0;

         O     #x_standby;
         O     #x_expansion;
         O     #x_compresion;
         A     #emer;
         BEC;
END_REGION

REGION Network 2: Plantilla de desconexión - STOP
   // Desconexión de la unidad productiva. 
   // Reinicia todos los parámetros para futuras conexiones.
   // Llamada a las maniobras usando la entrada asíncrona para indicar su pausa.
   // Después de la caja de código se especifica la instrucción “UN #start”, que coincide con la instrucción con la que se activó la plantilla. Esto es porque después de la caja, la RLO = 1 y /ER = 0. Por lo tanto, si la plantilla no se ejecuta, tras saltar la caja de código la RLO = 1 cuando debería ser 0 (UN #start no se cumple).
         AN    #start;
         R     #bit_trabajo;
         R     #bit_emer;
         R     #bit_error_config_expansion;
         R     #bit_error_config_compresion;
         R     #bit_error_tiempo_expansion;
         R     #bit_error_tiempo_compresion;
         R     #bit_standby;
         R     #bit_ocupacion;
         R     #temp_max;
         FR    #temp_max;

         JCN   stop;

         CALL  #SFC_Expansion
         ( sini             := ,
           sfin             := ,
           reset            := TRUE,
           tiempo_error     := ,
           temp_error       := ,
           bit_fin          := ,
           bit_error_tiempo := ,
           bit_error_config := ,
           bit_ocupacion    := ,
           actuador         := #expandir
         );


         CALL  #SFC_Compresion
         ( sini             := ,
           sfin             := ,
           reset            := TRUE,
           tiempo_error     := ,
           temp_error       := ,
           bit_fin          := ,
           bit_error_tiempo := ,
           bit_error_config := ,
           bit_ocupacion    := ,
           actuador         :=
         );

   stop: NOP   0;

         AN    #start;
         BEC;
END_REGION

REGION Network 3: Plantilla de conexión
   // Conexión de la unidad productiva.
         A     #start;
         FP    #bit_trabajo;
         S     #x_standby;
         R     #x_expansion;
         R     #x_compresion;
         R     #x_emer;
         R     #x_error_config_expansion;
         R     #x_error_config_compresion;
         R     #x_error_tiempo_expansion;
         R     #x_error_tiempo_compresion;
END_REGION

REGION Network 4: Plantilla de congelación
   // Congela la unidad productiva: habilitación de componentes y reset de actuadores.
   // Los estados no cambian y no se va a un estado especial, de forma que cuando se quite la congelación la unidad productiva vuelva a la etapa en la que estaba.
   // Se repite el estímulo de activación para saltar el resto de segmentos.
   // No se llama al actuador de compresión porque no existe.
         A     #cong;

         JCN   _cong;

         R     #temp_max;  //Habilitación de componentes
         FR    #temp_max;

         CALL  #SFC_Expansion
         ( sini             := ,
           sfin             := ,
           reset            := TRUE,
           tiempo_error     := ,
           temp_error       := ,
           bit_fin          := ,
           bit_error_tiempo := ,
           bit_error_config := ,
           bit_ocupacion    := ,
           actuador         := #expandir
         );

         CALL  #SFC_Compresion
         ( sini             := ,
           sfin             := ,
           reset            := TRUE,
           tiempo_error     := ,
           temp_error       := ,
           bit_fin          := ,
           bit_error_tiempo := ,
           bit_error_config := ,
           bit_ocupacion    := ,
           actuador         :=
         );

   _cong:NOP   0;

         A     #cong;  //Repetición del estímulo de activación
         BEC;
END_REGION

REGION Network 5: Salida del estado de emergencia
   // Rearme
         A     #x_emer;
         AN    #emer;
         A     #rearme;
         S     #x_standby;
         R     #x_emer;
END_REGION

REGION Network 6: Rearme errores síncronos
   // Se considera la posibilidad de rearme tras errores síncronos.
         O     #x_error_config_expansion;
         O     #x_error_config_compresion;
         O     #x_error_tiempo_expansion;
         O     #x_error_tiempo_compresion;
         A     #rearme;
         S     #x_standby;
         R     #x_error_config_expansion;
         R     #x_error_config_compresion;
         R     #x_error_tiempo_expansion;
         R     #x_error_tiempo_compresion;
END_REGION

REGION Network 7: x_standby -> x_expansion
         A     #x_standby;
         A     #push;
         S     #x_expansion;
         R     #x_standby;
END_REGION

REGION Network 8: Llamada a la maniobra de expansión
   // Entrada de error asíncrono false (se gestiona en la plantilla de desconexión).
         A     #x_expansion;

         JCN   _exp;
         CALL  #SFC_Expansion
         ( sini             := #scomp,
           sfin             := #sexp,
           reset            := FALSE,
           tiempo_error     := #tiempo_max,
           temp_error       := #temp_max,
           bit_fin          := #bit_fin_expansion,
           bit_error_tiempo := #bit_error_tiempo_expansion,
           bit_error_config := #bit_error_config_expansion,
           bit_ocupacion    := #bit_ocupacion,
           actuador         := #expandir
         );


         A     #bit_error_tiempo_expansion;
         S     #x_error_tiempo_expansion;
         R     #x_expansion;

         A     #bit_error_config_expansion;
         S     #x_error_config_expansion;
         R     #x_expansion;

         A     #bit_fin_expansion;
         S     #x_compresion;
         R     #x_expansion;

   _exp: NOP   0;
END_REGION

REGION Network 9: Llamada a la maniobra de compresión
   // No se indica actuador por ser un cilindro de simple efecto. Si no se actúa sobre el cilindro, este se comprime.
         A     #x_compresion;

         JCN   _comp;
         CALL  #SFC_Compresion
         ( sini             := #sexp,
           sfin             := #scomp,
           reset            := FALSE,
           tiempo_error     := #tiempo_max,
           temp_error       := #temp_max,
           bit_fin          := #bit_fin_compresion,
           bit_error_tiempo := #bit_error_tiempo_compresion,
           bit_error_config := #bit_error_config_compresion,
           bit_ocupacion    := #bit_ocupacion,
           actuador         :=
         );

         A     #bit_error_tiempo_compresion;
         S     #x_error_tiempo_compresion;
         R     #x_compresion;

         A     #bit_error_config_compresion;
         S     #x_error_config_compresion;
         R     #x_compresion;

         A     #bit_fin_compresion;
         S     #x_standby;
         R     #x_compresion;

   _comp:NOP   0;
END_REGION

REGION Network 10: Bit de standby
   // Indica el estado de standby.
         A     #x_standby;
         =     #bit_standby;
END_REGION

REGION Network 11: Bit de emergencia
   // Indica el estado de emergencia.
         A     #x_emer;
         =     #bit_emer;
END_REGION

REGION Network 12: Bit error tiempo expansión
   // Indica el estado de error síncrono por tiempo de expansión.
         A     #x_error_tiempo_expansion;
         =     #bit_error_tiempo_expansion;
END_REGION

REGION Network 13: Bit error tiempo compresión
   // Indica el estado de error síncrono por tiempo de compresión.
         A     #x_error_tiempo_compresion;
         =     #bit_error_tiempo_compresion;
END_REGION

REGION Network 14: Bit error config expansión
   // Indica el estado de error síncrono por mala configuración inicial en la expansión.
         A     #x_error_config_expansion;
         =     #bit_error_config_expansion;
END_REGION

REGION Network 15: Bit error config compresión
   // Indica el estado de error síncrono por mala configuración inicial en la compresión.
         A     #x_error_config_compresion;
         =     #bit_error_config_compresion;
END_REGION
END_FUNCTION_BLOCK

// folder: Emergencia

FUNCTION_BLOCK "GEMER_Local"   // FB5, STL
TITLE = Grafcet de emergencia local robot
{ S7_Optimized_Access := 'TRUE' }
VERSION : 0.1
// Se encarga de forzar al estado de emergencia a las unidades productivas a las que controle. Se ha implementado en un FB porque tiene estados internos locales (los estados de GEMER_Global son globales y, además, es requisito del trabajo implementar dicho bloque como FC sin parámetros). 
// Se reutilizará esta función con cada una de las unidades productivas, con la diferencia de que se llamará cada vez a un bloque de datos diferente.
// Presenta la siguiente interfaz:
// - Emer: informa de emergencia global o local.
// - Rearme: rearme global o local.
// - Bit_emer: informa que la función se encuentra en estado de emergencia.
// - X_marcha: estado de marcha.
// - X_emer: estado de emergencia.
// - Bit_trabajo: controla la conexión del bloque.
   VAR_INPUT
      emer : Bool;
      rearme : Bool;
   END_VAR
   VAR_OUTPUT
      bit_emer : Bool;
   END_VAR
   VAR
      x_marcha : Bool;
      x_emer : Bool;
      bit_trabajo : Bool;
   END_VAR
BEGIN

REGION Network 1: Plantilla de conexión
   // Solamente se ejecuta una vez (la función no se desconecta) con el inicio del programa (OB100).
         SET;
         FP    #bit_trabajo;
         S     #x_marcha;
         R     #x_emer;
END_REGION

REGION Network 2: Plantilla de forzado - Emergencia
         A     #emer;
         S     #x_emer;
         R     #x_marcha;
         =     #bit_emer;
         BEC;
END_REGION

REGION Network 3: x_marcha -> x_emer
         A     #x_marcha;
         A     #emer;
         S     #x_emer;
         R     #x_marcha;
END_REGION

REGION Network 4: x_emer -> x_marcha
         A     #x_emer;
         AN    #emer;
         A     #rearme;
         S     #x_marcha;
         R     #x_emer;
END_REGION

REGION Network 5: Tratamiento estado de emergencia
         A     #x_emer;
         =     #bit_emer;
END_REGION
END_FUNCTION_BLOCK

FUNCTION "GEMER_Global" : Void   // FC6, STL
TITLE = Emergencia global
{ S7_Optimized_Access := 'TRUE' }
VERSION : 0.1
// Se encarga de coordinar la emergencia global en toda la celda, llamando a los bloques de emergencia locales. Usa variables absolutas (FC sin parámetros y que controla estados globales).  Se inicia directamente en estado de marcha con el OB100.
BEGIN

REGION Network 1: x_marcha -> x_emer
         A     "x_marcha";
         A     "emer";
         S     "x_emer";
         R     "x_marcha";
END_REGION

REGION Network 2: x_emer -> x_marcha
         A     "x_emer";
         AN    "emer";
         A     "rearme";
         S     "x_marcha";
         R     "x_emer";

         JCN   _rearme;

         CALL  "GEMER_Local", "GEMER_Robot1_DB"
         ( emer     := FALSE,
           rearme   := TRUE,
           bit_emer := "robot1_emer"
         );

         CALL  "GEMER_Local", "GEMER_Robot2_DB"
         ( emer     := FALSE,
           rearme   := TRUE,
           bit_emer := "robot2_emer"
         );

         CALL  "GEMER_Local", "GEMER_CNC1_DB"
         ( emer     := FALSE,
           rearme   := TRUE,
           bit_emer := "cnc1_emer"
         );

         CALL  "GEMER_Local","GEMER_CNC2_DB"
         ( emer     := FALSE,
           rearme   := TRUE,
           bit_emer := "cnc2_emer"
         );

         CALL  "GEMER_Local","GEMER_Simple_Efecto1_DB"
         ( emer     := FALSE,
           rearme   := TRUE,
           bit_emer := "sef1_emer"
         );

   _rearme:NOP   0;
END_REGION

REGION Network 3: Emergencia
         A     "x_emer";

         JCN   _emergencia;

         CALL  "GEMER_Local","GEMER_Robot1_DB"
         ( emer     := TRUE,
           rearme   := FALSE,
           bit_emer := "robot1_emer"
         );

         CALL  "GEMER_Local", "GEMER_Robot2_DB"
         ( emer     := TRUE,
           rearme   := FALSE,
           bit_emer := "robot2_emer"
         );

         CALL  "GEMER_Local", "GEMER_CNC1_DB"
         ( emer     := TRUE,
           rearme   := FALSE,
           bit_emer := "cnc1_emer"
         );

         CALL  "GEMER_Local","GEMER_CNC2_DB"
         ( emer     := TRUE,
           rearme   := FALSE,
           bit_emer := "cnc2_emer"
         );

         CALL  "GEMER_Local","GEMER_Simple_Efecto1_DB"
         ( emer     := TRUE,
           rearme   := FALSE,
           bit_emer := "sef1_emer"
         );

         CALL  "GMM", "GMM_DB"
         ( on              := ,
           lote_pequenio   := ,
           lote_mediano    := ,
           lote_grande     := ,
           mcong           := ,
           cong            := ,
           emer            := TRUE,
           bit_paro        := "gmm_bit_paro",
           bit_marcha      := "gmm_bit_marcha",
           bit_congelacion := "gmm_bit_congelacion"
         );

   _emergencia:NOP   0;
END_REGION
END_FUNCTION

// folder: Maniobras

FUNCTION_BLOCK "SFC_Programa"   // FB1, STL
TITLE = Programas unidad productiva
{ S7_Optimized_Access := 'TRUE' }
VERSION : 0.1
// Ejecuta los programas de la unidad productiva con control de tiempo y configuración inicial.
// Tiene los siguientes parámetros:
// - sensor1: receptividad entre xe y x1.
// - sensor2: receptividad entre xs y x1.
// - reset: indica la desconexión por error asíncrono.
// - tiempo_error: tiempo límite antes de error síncrono.
// - temp_error: temporizador de error síncrono.
// - bit_fin: la maniobra ha finalizado correctamente.
// - bit_error_tiempo: tiempo límite agotado (error síncrono).
// - bit_error_config: mala configuración inicial (error síncrono).
// - bit_ocupacion: maniobra en ejecución.
// - actuador1: programa a cargar en el robot.
// - bit_trabajo: conecta el bloque maniobra.
// - xe: estado inicial.
// - x1: estado de ejecución del programa.
// - x2: estado de error síncrono por tiempo.
// - x3: estado de error síncrono por mala configuración inicial.
// - xs: estado final.
// - mf_sensor2: marca de flanco del sensor 2.
// - mp_sensor2: merca de pulso del sensor 2.
   VAR_INPUT
      sensor1 : Bool;
      sensor2 : Bool;
      reset : Bool;
      tiempo_error : S5Time := S5T#10S;
      temp_error : Timer;
   END_VAR
   VAR_OUTPUT
      bit_fin : Bool;
      bit_error_tiempo : Bool;
      bit_error_config : Bool;
      bit_ocupacion : Bool;
      actuador1 : Bool;
   END_VAR
   VAR
      xe : Bool;
      x1 : Bool;
      x2 : Bool;
      x3 : Bool;
      xs : Bool;
      bit_trabajo : Bool;
      mf_sensor2 : Bool;
   END_VAR
   VAR_TEMP
      mp_sensor2 : Bool;
   END_VAR
BEGIN

REGION Network 1: Plantilla de desconexión - error asíncrono
   // Desconexión en caso de error asíncrono (actuadores, temporizadores, bit de fin y bit de trabajo)
         A     #reset;
         R     #bit_fin;
         R     #bit_trabajo;  //Futuros arranques
         R     #bit_ocupacion;
         R     #actuador1;
         R     #temp_error;  //Habilitación de temporizadores
         FR    #temp_error;
         R     #mf_sensor2;
         BEC;
END_REGION

REGION Network 2: Error síncrono por tiempo
   // Desconexión por tiempo límite (actuadores, temporizadores, bit de fin y bit de trabajo). 
   // Es necesario desconectar x2 porque si no no se podría volver a ejecutar la maniobra (se saldría continuamente
   // del bloque).
   // Se deja todo preparado para futuras conexiones.
         A     #x2;
         S     #bit_error_tiempo;
         R     #x2;
         R     #bit_fin;
         R     #bit_trabajo;  //Futuros arranques
         R     #bit_ocupacion;
         R     #actuador1;
         R     #temp_error;  // Habilitación de temporizadores
         FR    #temp_error;
         R     #mf_sensor2;
         BEC;
END_REGION

REGION Network 3: Error síncrono por mala configuración inicial
   // Desconexión por mala configuración inicial.
   // Es necesario desconectar x3 porque si no no se podría volver a ejectar la maniobra.
   // Se deja todo preparado para futuras conexiones.
         A     #x3;
         S     #bit_error_config;
         R     #x3;
         R     #bit_trabajo;
         R     #bit_fin;
         R     #bit_ocupacion;
         R     #actuador1;
         R     #temp_error;
         FR    #temp_error;
         R     #mf_sensor2;
         BEC;
END_REGION

REGION Network 4: Plantilla de desconexión - final de maniobra
   // Desconexión por fin de la maniobra
         A     #xs;
         S     #bit_fin;
         R     #xs;
         R     #bit_trabajo;
         R     #bit_ocupacion;
         R     #actuador1;
         R     #temp_error;
         FR    #temp_error;
         R     #mf_sensor2;
         BEC;
END_REGION

REGION Network 5: Plantilla de conexión
   // Inicialización del bloque a valores iniciales.
   // Se resetean los bits de control.
         SET;
         FP    #bit_trabajo;
         R     #bit_fin;
         R     #bit_error_config;
         R     #bit_error_tiempo;
         R     #bit_ocupacion;
         S     #xe;
         R     #x1;
         R     #x2;
         R     #x3;
         R     #xs;
END_REGION

REGION Network 6: Configuración flancos
   // Sensor 2 representa la señal home.
   // La maniobra comienza con el robot en home y termina con el robot en home. 
   // Se produce un flanco de la señal home (si se gestiona por nivel la maniobra de 
   // carga duraría tan solo un ciclo).
         A     #sensor2;
         FP    #mf_sensor2;
         =     #mp_sensor2;
END_REGION

REGION Network 7: Configuración temporizador maniobra
   // Carga el temporizador que establece el tiempo para llevar a cabo la maniobra.
   // Temporizador se (vigila el tiempo en el estado actual).
         A     #x1;
         L     #tiempo_error;
         SD    #temp_error;
END_REGION

REGION Network 8: x1 -> x2 (Error síncrono por tiempo)
   // Tiempo límite agotado
         A     #x1;
         A     #temp_error;
         S     #x2;
         R     #x1;
END_REGION

REGION Network 9: x1 -> xs - Estado fugaz
   // Al entrar a la maniobra se produce una marca de pulso si la configuración inicial es correcta: "sensor2" está a nivel alto y la marca de flanco comienza el bloque siempre a nivel bajo. Esto provocaría que la maniobra sea fugaz.
   // Se cambia el orden de las etapas para arreglar este problema.
         A     #x1;
         A     #mp_sensor2;
         S     #xs;
         R     #x1;
END_REGION

REGION Network 10: xe -> x3 (Error síncrono por mala configuración inicial)
   // El sensor 1 representa la señal que activa el programa del robot.
   // El sensor 2 representa la señal home.
   // Cuando se inicia la maniobra el robot debe estar en home y la señal del programa
   // tiene que estar activa.
   // El error es prioritario ante la transición a la ejecución del programa.
         ON    #sensor1;
         ON    #sensor2;
         A     #xe;
         S     #x3;
         R     #xe;
END_REGION

REGION Network 11: xe -> x1
         A     #xe;
         A     #sensor1;
         A     #sensor2;
         S     #x1;
         R     #xe;
END_REGION

REGION Network 12: Cargar programa
         A     #x1;
         =     #actuador1;
         =     #bit_ocupacion;
END_REGION
END_FUNCTION_BLOCK

FUNCTION_BLOCK "SFC_Cilindro"   // FB3, STL
TITLE = Maniobras del cilindro (expansión y compresión)
{ S7_Optimized_Access := 'TRUE' }
VERSION : 0.1
// Se encarga de ejecutar las maniobras de carga y descarga de la unidad productiva.
// Tiene los siguientes parámetros:
// - sini: estado inicial del cilindro.
// - sfin: estado final del cilindro.
// - reset: indica la desconexión por error asíncrono.
// - tiempo_error: tiempo límite antes de error síncrono.
// - temp_error: temporizador de error síncrono.
// - bit_fin: la maniobra ha finalizado correctamente.
// - bit_error_tiempo: tiempo límite agotado (error síncrono).
// - bit_error_config: mala configuración inicial (error síncrono).
// - bit_ocupacion: la unidad productiva está ejecutando la maniobra (x1)
// - actuador: programa a cargar en el robot.
// - bit_trabajo: conecta el bloque maniobra.
// - xe: estado inicial.
// - x1: estado de ejecución del programa.
// - x2: estado de error síncrono por tiempo.
// - x3: estado de error síncrono por mala configuración inicial.
// - xs: estado final.
   VAR_INPUT
      sini : Bool;
      sfin : Bool;
      reset : Bool;
      tiempo_error : S5Time;
      temp_error : Timer;
   END_VAR
   VAR_OUTPUT
      bit_fin : Bool;
      bit_error_tiempo : Bool;
      bit_error_config : Bool;
      bit_ocupacion : Bool;
      actuador : Bool;
   END_VAR
   VAR
      xe : Bool;
      x1 : Bool;
      x2 : Bool;
      x3 : Bool;
      xs : Bool;
      bit_trabajo : Bool;
   END_VAR
BEGIN

REGION Network 1: Plantilla de desconexión - error asíncrono
   // Desconexión en caso de error asíncrono (actuadores, temporizadores, bit de fin y bit de trabajo)
         A     #reset;
         R     #bit_fin;
         R     #bit_trabajo;  //Futuros arranques
         R     #bit_ocupacion;
         R     #actuador;
         R     #temp_error;  //Habilitación de temporizadores
         FR    #temp_error;
         BEC;
END_REGION

REGION Network 2: Error síncrono por tiempo
   // Desconexión por tiempo límite (actuadores, temporizadores, bit de fin y bit de trabajo). 
   // Es necesario desconectar x2 porque si no no se podría volver a ejecutar la maniobra (se saldría continuamente
   // del bloque).
   // Se deja todo preparado para futuras conexiones.
         A     #x2;
         S     #bit_error_tiempo;
         R     #x2;
         R     #bit_fin;
         R     #bit_trabajo;  //Futuros arranques
         R     #bit_ocupacion;
         R     #actuador;
         R     #temp_error;  // Habilitación de temporizadores
         FR    #temp_error;
         BEC;
END_REGION

REGION Network 3: Error síncrono por mala configuración inicial
   // Desconexión por mala configuración inicial.
   // Es necesario desconectar x3 porque si no no se podría volver a ejectar la maniobra.
   // Se deja todo preparado para futuras conexiones.
         A     #x3;
         S     #bit_error_config;
         R     #x3;
         R     #bit_trabajo;
         R     #bit_fin;
         R     #bit_ocupacion;
         R     #actuador;
         R     #temp_error;
         FR    #temp_error;
         BEC;
END_REGION

REGION Network 4: Plantilla de desconexión - final de maniobra
   // Desconexión por fin de la maniobra
         A     #xs;
         S     #bit_fin;
         R     #xs;
         R     #bit_trabajo;
         R     #bit_ocupacion;
         R     #actuador;
         R     #temp_error;
         FR    #temp_error;
         BEC;
END_REGION

REGION Network 5: Plantilla de conexión
   // Inicialización del bloque a valores iniciales.
   // Se resetean los bits de control.
         SET;
         FP    #bit_trabajo;
         R     #bit_fin;
         R     #bit_error_config;
         R     #bit_error_tiempo;
         R     #bit_ocupacion;
         S     #xe;
         R     #x1;
         R     #x2;
         R     #x3;
         R     #xs;
END_REGION

REGION Network 6: Configuración temporizador maniobra
   // Carga el temporizador que establece el tiempo para llevar a cabo la maniobra.
   // Temporizador se (vigila el tiempo en el estado actual).
         A     #x1;
         L     #tiempo_error;
         SD    #temp_error;
END_REGION

REGION Network 7: xe -> x3 (Error síncrono por mala configuración inicial)
   // Si el cilindro no se encuentra en la posición inicial (expandido o contraído, según la maniobra) o
   // si se encuentra en la posición final, la configuración inicial es incorrecta.
         ON    #sini;
         O     #sfin;
         A     #xe;
         S     #x3;
         R     #xe;
END_REGION

REGION Network 8: xe -> x1
         A     #xe;
         A     #sini;
         S     #x1;
         R     #xe;
END_REGION

REGION Network 9: x1 -> xs
         A     #x1;
         A     #sfin;
         S     #xs;
         R     #x1;
END_REGION

REGION Network 10: x1 -> x2 (Error síncrono por tiempo)
   // Tiempo límite agotado
         A     #x1;
         A     #temp_error;
         S     #x2;
         R     #x1;
END_REGION

REGION Network 11: Acción (expandir o comprimir)
         A     #x1;
         =     #actuador;
         =     #bit_ocupacion;
END_REGION
END_FUNCTION_BLOCK

// folder: Modos de marcha

FUNCTION_BLOCK "GMM"   // FB7, STL
TITLE = Grafcet modos de marcha
{ S7_Optimized_Access := 'TRUE' }
VERSION : 0.1
// Se encarga de determinar los modos de marcha (lote pequeño, lote mediano, lote grande o congelación). Cuando se encuentra en marcha las unidades productivas están activas; cuando está en parada se desconectan. Se inicia con el OB100 y permanece siempre activo. Presenta la siguiente interfaz:
// - On: pasa al estado de marcha.
// - Lote_pequenio: los lotes a procesar son pequeños.
// - Lote_mediano: los lotes a procesar son medianos.
// - Lote grande: los lotes a procesar son grandes.
// - Mcong: modo de marcha con congelación.
// - Cong: señal de congelación.
// - Emer: señal de emergencia.
// - Bit_paro: indica que el bloque se encuentra en paro.
// - Bit_marcha: indica que el bloque está en marcha (si no está en parada).
// - Bit_congelacion: indica que el bloque está en estado de congelación.
// - X_parada: estado de parada.
// - X_marcha: estado de marcha.
// - X_lote_pequenio: estado de producción de lotes pequeños.
// - X_lote_mediano: estado de producción de lotes medianos.
// - X_lote_grande: estado de producción de lotes grandes.
// - X_mcong: estado de marcha con posibilidad de congelación.
// - X_cong: estado de congelación.
// - Bit_trabajo: controla la conexión del bloque.
   VAR_INPUT
      on : Bool;
      lote_pequenio : Bool;
      lote_mediano : Bool;
      lote_grande : Bool;
      mcong : Bool;
      cong : Bool;
      emer : Bool;
   END_VAR
   VAR_OUTPUT
      bit_paro : Bool;
      bit_marcha : Bool;
      bit_congelacion : Bool;
   END_VAR
   VAR
      x_parada : Bool;
      x_marcha : Bool;
      x_lote_pequenio : Bool;
      x_lote_mediano : Bool;
      x_lote_grande : Bool;
      x_mcong : Bool;
      x_cong : Bool;
      bit_trabajo : Bool;
   END_VAR
BEGIN

REGION Network 1: Plantilla de conexión
   // Conecta el bloque con el inicio del programa en el OB100. Solo se ejecuta una vez la plantilla de conexión.
         SET;
         FP    #bit_trabajo;
         S     #x_parada;
         R     #x_marcha;
         R     #x_lote_pequenio;
         R     #x_lote_mediano;
         R     #x_lote_grande;
         R     #x_cong;
END_REGION

REGION Network 2: Plantilla de forzado - Error asíncrono
   // En caso de emergencia global, se fuerza al estado de parada y se reinician los demás estados.
         A     #emer;
         S     #x_parada;
         R     #x_marcha;
         R     #x_lote_grande;
         R     #x_lote_mediano;
         R     #x_lote_pequenio;
         R     #x_mcong;
         R     #x_cong;
         R     #bit_marcha;
         R     #bit_congelacion;
         BEC;
END_REGION

REGION Network 3: x_parada -> x_marcha
         A     #x_parada;
         A     #on;
         S     #x_marcha;
         R     #x_parada;
END_REGION

REGION Network 4: x_marcha -> x_parada
         A     #x_marcha;
         A     "cnc1_b_standby";
         A     "cnc2_b_standby";
         A     "robot1_b_standby";
         A     "robot2_b_standby";
         A     "sef1_b_standby";
         AN    #on;
         S     #x_parada;
         R     #x_marcha;
END_REGION

REGION Network 5: x_marcha -> x_lote_pequenio
         A     #x_marcha;
         A     #lote_pequenio;
         S     #x_lote_pequenio;
         R     #x_marcha;
END_REGION

REGION Network 6: x_marcha -> x_lote_mediano
         A     #x_marcha;
         A     #lote_mediano;
         S     #x_lote_mediano;
         R     #x_marcha;
END_REGION

REGION Network 7: x_marcha -> x_lote_grande
         A     #x_marcha;
         A     #lote_grande;
         S     #x_lote_grande;
         R     #x_marcha;
END_REGION

REGION Network 8: x_marcha -> x_mcong
         A     #x_marcha;
         A     #mcong;
         S     #x_mcong;
         R     #x_marcha;
END_REGION

REGION Network 9: x_mcong -> x_cong
         A     #x_mcong;
         A     #cong;
         S     #x_cong;
         R     #x_mcong;
END_REGION

REGION Network 10: x_lote_pequenio -> x_marcha
         A     #x_lote_pequenio;
         AN    #lote_pequenio;
         S     #x_marcha;
         R     #x_lote_pequenio;
END_REGION

REGION Network 11: x_lote_mediano -> x_marcha
         A     #x_lote_mediano;
         AN    #lote_mediano;
         S     #x_marcha;
         R     #x_lote_mediano;
END_REGION

REGION Network 12: x_lote_grande-> x_marcha
         A     #x_lote_grande;
         AN    #lote_grande;
         S     #x_marcha;
         R     #x_lote_grande;
END_REGION

REGION Network 13: x_cong -> x_marcha
         A     #x_cong;
         AN    #mcong;
         AN    #cong;
         S     #x_marcha;
         R     #x_cong;
END_REGION

REGION Network 14: x_cong -> x_mcong
         A     #x_cong;
         AN    #cong;
         S     #x_mcong;
         R     #x_cong;
END_REGION

REGION Network 15: Tratamiento lote pequeño
   // Carga los datos de producción para lotes pequeños.
         A     #x_lote_pequenio;

         JCN   _lotePequenio;

         L     "datosLotePequenio".tmax_cnc_lapiz;
         T     "datosProduccion".tmax_cnc_lapiz;
         L     "datosLotePequenio".tmax_cnc_sacapuntas;
         T     "datosProduccion".tmax_cnc_sacapuntas;
         L     "datosLotePequenio".tmax_cnc_escuadra;
         T     "datosProduccion".tmax_cnc_escuadra;
         L     "datosLotePequenio".tmax_cnc_cartabon;
         T     "datosProduccion".tmax_cnc_cartabon;

   _lotePequenio:NOP   0;
END_REGION

REGION Network 16: Tratamiento lote mediano
   // Carga los datos de producción para lotes medianos.
         A     #x_lote_mediano;

         JCN   _loteMediano;

         L     "datosLoteMediano".tmax_cnc_lapiz;
         T     "datosProduccion".tmax_cnc_lapiz;
         L     "datosLoteMediano".tmax_cnc_sacapuntas;
         T     "datosProduccion".tmax_cnc_sacapuntas;
         L     "datosLoteMediano".tmax_cnc_escuadra;
         T     "datosProduccion".tmax_cnc_escuadra;
         L     "datosLoteMediano".tmax_cnc_cartabon;
         T     "datosProduccion".tmax_cnc_cartabon;

   _loteMediano:NOP   0;
END_REGION

REGION Network 17: Tratamiento lote grande
   // Carga los datos de producción para lotes grandes.
         A     #x_lote_grande;

         JCN   _loteGrande;

         L     "datosLoteGrande".tmax_cnc_lapiz;
         T     "datosProduccion".tmax_cnc_lapiz;
         L     "datosLoteGrande".tmax_cnc_sacapuntas;
         T     "datosProduccion".tmax_cnc_sacapuntas;
         L     "datosLoteGrande".tmax_cnc_escuadra;
         T     "datosProduccion".tmax_cnc_escuadra;
         L     "datosLoteGrande".tmax_cnc_cartabon;
         T     "datosProduccion".tmax_cnc_cartabon;

   _loteGrande:NOP   0;
END_REGION

REGION Network 18: Bit de marcha
         AN    #x_parada;
         =     #bit_marcha;
END_REGION

REGION Network 19: Bit de parada
         A     #x_parada;
         =     #bit_paro;
END_REGION

REGION Network 20: Bit de congelación
         A     #x_cong;
         =     #bit_congelacion;
END_REGION
END_FUNCTION_BLOCK

// folder: Palets vacíos

FUNCTION_BLOCK "UP_Palets_Vacios"   // FB2, STL
TITLE = Gestión palets vacíos
{ S7_Optimized_Access := 'TRUE' }
VERSION : 0.1
// Funciona como interfaz para conocer el estado de la pila de palets. Se sirve de la función alturaPalets. Tiene los siguientes parámetros:
// - start: conecta y desconecta la unidad productiva.
// - Emer: entra en estado de emergencia.
// - Rearme: sale del estado de emergencia.
// - Cong: entra en congelación.
// - Hraw: señal de entrada analógica muestreada que representa la altura de la pila de palets vacíos.
// - LO_LIM: límite mínimo de altura para la interpolación.
// - HI_LIM: límite máximo de altura para la interpolación.
// - Hmin: altura mínima (magnitud física) de la pila de palets vacíos para ser recogida.
// - Hmax: altura máxima (magnitud física) de la pila de palets vacíos para saturarse (no se pueden colocar más palets sobre la misma).
// - Recoger_pila: llamada a los AGVs para recoger la pila de palets vacíos.
// - Pila_saturada: llamada a los AGVs para recoger la pila de palets vacíos (urgentemente).
// - Error_medida: la magnitud medida está fuera de rango (LO_LIM – HI_LIM).
// - H_real: altura de la pila de palets vacíos en forma física.
// - H>hmin: conector indicando que la altura de la pila de palets es mayor que h_min.
// - H<hmin: conector indicando que la altura de la pila de palets es menor que h_min.
// - H>hmax: conector indicando que la altura de la pila de palets es mayor que h_max.
// - X1: estado de standby.
// - X2: estado indicando que la altura de la pila de palets vacíos es mayor que hmin.
// - X3: estado indicando que la altura de la pila de palets vacíos es mayor que hmax.
// - X_emer: estado de emergencia.
// - Bit_trabajo: bit de control del encendido de la unidad productiva (flanco positivo de start).
// - Bit_standby: bit indicando el estado de standby.
// - Bit_emer: bit indicando el estado de emergencia.
   VAR_INPUT
      start : Bool;
      emer : Bool;
      rearme : Bool;
      cong : Bool;
      hraw : Int;
      LO_LIM : Real;
      HI_LIM : Real;
      hmin : Real;
      hmax : Real;
   END_VAR
   VAR_OUTPUT
      recoger_pila : Bool;
      pila_saturada : Bool;
      error_medida : Bool;
      h_real : Real;
   END_VAR
   VAR_IN_OUT
      "h>hmin" : Bool;
      "h>hmax" : Bool;
      "h<hmin" : Bool;
   END_VAR
   VAR
      x1 : Bool;
      x2 : Bool;
      x3 : Bool;
      x_emer : Bool;
      bit_trabajo : Bool;
      bit_standby : Bool;
      bit_emer : Bool;
   END_VAR
BEGIN

REGION Network 1: Plantilla de desconexión - Error asíncrono
   // Entra en error asíncrono por emergencia. Desconecta las salidas y activa el estado de emergencia.
         A     #emer;
         S     #x_emer;
         R     #recoger_pila;
         R     #pila_saturada;
         R     #bit_standby;
         R     #error_medida;
         R     #"h<hmin";
         R     #"h>hmax";
         R     #"h>hmin";
         =     #bit_emer;
         BEC;
END_REGION

REGION Network 2: Plantilla de desconexión - STOP
   // Se activa al desconectar la unidad productiva. Resetea los bits de control (importante resetear el bit de trabajo para futuras conexiones) y las salidas.
         AN    #start;
         R     #bit_trabajo;
         R     #bit_standby;
         R     #recoger_pila;
         R     #pila_saturada;
         R     #error_medida;
         R     #"h<hmin";
         R     #"h>hmax";
         R     #"h>hmin";
         BEC;
END_REGION

REGION Network 3: Plantilla de conexión
   // Conecta la unidad productiva por flanco positivo del bit de trabajo (debe ser reseteado adecuadamente después de la desconexión). Establece el estado de standby como estado inicial.
         A     #start;
         FP    #bit_trabajo;
         S     #x1;
         R     #x2;
         R     #x3;
         R     #x_emer;
END_REGION

REGION Network 4: Plantilla de congelación
   // Resetea las salidas y mantiene el estado actual en el que estaba para poder seguir produciendo tras descongelar.
         A     #cong;
         R     #recoger_pila;
         R     #pila_saturada;
         R     #error_medida;
         R     #"h<hmin";
         R     #"h>hmax";
         R     #"h>hmin";
         BEC;
END_REGION

REGION Network 5: Salida de emergencia
   // Rearme desde el estado de emergencia.
         A     #x_emer;
         AN    #emer;
         A     #rearme;
         S     #x1;
         R     #x_emer;
END_REGION

REGION Network 6: Llamada a altura palets
   // Llama al FC alturaPalets para conocer la altura de la pila de palets, así como los conectores usados para la transición entre estados (h<hmin, h>hmin, h>hmax). Los datos de los valores extremos, así como de hmin y hmax están en el DB datosProduccion.
         CALL  "alturaPalets"
         ( RAW       := #hraw,
           BIPOLAR   := FALSE,
           LO_LIM    := #LO_LIM,
           HI_LIM    := #HI_LIM,
           h_min     := #hmin,
           h_max     := #hmax,
           reset     := FALSE,
           REAL_VAL  := #h_real,
           "h>h_min" := #"h>hmin",
           "h>h_max" := #"h>hmax",
           "h<h_min" := #"h<hmin",
           error     := #error_medida
         );
END_REGION

REGION Network 7: x1 -> x2
         A     #x1;
         A     #"h>hmin";
         S     #x2;
         R     #x1;
END_REGION

REGION Network 8: x1 -> x3
         A     #x1;
         A     #"h>hmax";
         S     #x3;
         R     #x1;
END_REGION

REGION Network 9: x2 -> x1
         A     #x2;
         A     #"h<hmin";
         S     #x1;
         R     #x2;
END_REGION

REGION Network 10: x3 -> x1
         A     #x3;
         A     #"h<hmin";
         S     #x1;
         R     #x3;
END_REGION

REGION Network 11: Recoger pila
         A     #x2;
         =     #recoger_pila;
END_REGION

REGION Network 12: Pila saturada
         A     #x3;
         =     #pila_saturada;
END_REGION
END_FUNCTION_BLOCK

FUNCTION "alturaPalets" : Void   // FC7, STL
TITLE = Gestión altura pila palets vacíos
{ S7_Optimized_Access := 'TRUE' }
VERSION : 0.1
// Gestiona las señales analógicas de la pila de palets vacíos.
// Devuelve los conectores con las condiciones necesarias para la implemetación del grafcet.
// Toma los siguientes parámetros:
// - RAW: señal analógica muestreada.
// - BIPOLAR: especifica si la señal puede tomar valores en un rango solo positivo o positivo y negativo.
// - LO_LIM: altura mínima permitida para la interpolación.
// - HI_LIM: altura máxima permitida para la interpolación.
// - h_min: altura mínima de la pila de palets para ser transportada a otro lugar de la fábrica. Se pueden apilar más palets en la pila después de alcanzar este valor.
// - h_max: altura máxima de la pila de palets para ser transportada a otro lugar de la fábrica. No se pueden apilar más palets en la pila si se alcanza este valor.
// - reset: desconecta el bloque FC.
// - REAL_VAL: valor de la magnitud física (altura).
// - h>h_min: la altura de la pila ha superado h_min.
// - h>h_max: la altura de la pila ha superado h_max.
// - h<h_min: la altura de la pila es menor que h_min.
// - error: la altura medida está fuera de límites.
   VAR_INPUT
      RAW : Int;
      BIPOLAR : Bool;
      LO_LIM : Real;
      HI_LIM : Real;
      h_min : Real;
      h_max : Real;
      reset : Bool;
   END_VAR
   VAR_OUTPUT
      REAL_VAL : Real;
      "h>h_min" : Bool;
      "h>h_max" : Bool;
      "h<h_min" : Bool;
      error : Bool;
   END_VAR
   VAR_TEMP
      ret_val_1 : Word;
   END_VAR
BEGIN

REGION Network 1: Plantilla de desconexión
   // Resetea las salidas
         A     #reset;
         R     #"h>h_min";
         R     #"h>h_max";
         R     #"h<h_min";
         R     #error;
         BEC;
END_REGION

REGION Network 2: Llamada a la función SCALE
   // Convierte la señal muestreada (raw) en señal física (real_val)
         CALL  SCALE
         ( IN      := #RAW,
           HI_LIM  := #HI_LIM,
           LO_LIM  := #LO_LIM,
           BIPOLAR := #BIPOLAR,
           RET_VAL := #ret_val_1,
           OUT     := #REAL_VAL
         );
END_REGION

REGION Network 3: Error límites
   // Devuelve error si la señal está fuera de los límites hi_lim y lo_lim
   // Código de error: W#16#0008
   // Error = true si ret_val_err = código de error
         L     #ret_val_1;
         L     W#16#0008;
         ==I;
         =     #error;
END_REGION

REGION Network 4: h > h_min
   // Conector "h > h_min"
         L     #REAL_VAL;  //ACU2
         L     #h_min;  //ACU1
         >R;
         =     #"h>h_min";
END_REGION

REGION Network 5: h < h_min
   // Conector "h < h_min"
         A     <0;
         =     #"h<h_min";
END_REGION

REGION Network 6: h > h_max
   // Conector "h > h_max"
         L     #REAL_VAL;  // ACU2
         L     #h_max;  // ACU1
         >R;
         =     #"h>h_max";
END_REGION
END_FUNCTION

// folder: Robots carga / descarga

FUNCTION_BLOCK "UP_Robot"   // FB4, STL
TITLE = Unidad productiva robot pick and place
{ S7_Optimized_Access := 'TRUE' }
VERSION : 0.1
// Gestiona el robot pick and place.
// Presenta los siguientes parámetros:
// - start: inicia la unidad productiva.
// - emer: señal de emergencia (error asíncrono).
// - cong: señal de congelación.
// - rearme: vuelta al estado de standby de un estado de error.
// - dc: señal de carga.
// - fin_p: señal de descarga.
// - home: indica el estado en la posición fetal.
// - tiempo_max: tiempo máximo para las maniobras.
// - temp_max: temporizador de las manioabras.
// - cargar: programa de carga.
// - descargar: programa de descarga.
// - bit_standby: estado de standby.
// - bit_ocupación: el robot se encuentra en medio de una maniobra.
// - bit_error_tiempo_carga: error síncrono en la carga.
// - bit_error_tiempo_descarga: error síncrono en la descarga.
// - bit_error_config_carga: error síncrono por mala configuración inicial en la carga.
// - bit_error_config_descarga: error síncrono por mala configuración inicial en la descarga.
// - bit_emer: estado de emergencia.
// - bit_trabajo: se encarga de la conexión de la unidad productiva.
// - x_carga: estado de carga.
// - x_descarga: estado de descarga.
// - x_standby: estado de standby.
// - x_error_tiempo_carga: estado de error síncrono en la carga.
// - x_error_tiempo_descarga: estado de error síncrono en la descarga.
// - x_error_config_carga: estado de error síncrono por mala configuración inicial en la carga.
// - x_error_config_descarga: estado de error síncrono por mala configuración inicial en la descarga.
// - x_espera_home_carga: estado transitorio entre la maniobra de carga y el estado de standby.
// - x_espera_home_descarga: estado transitorio entre la maniobra de descarga y el estado de standby.
// - SFC_Programa_Carga: maniobra de carga de tipo SFC_Programa con bloque de datos multiinstancia.
// - SFC_Programa_ Descarga: maniobra de descarga de tipo SFC_Programa con bloque de datos multiinstancia.
// - bit_fin_carga: finalización de la carga.
// - bit_fin_descarga: finalización de la descarga. 
// 
// Las variables "bit_fin_carga" y "bit_fin_descarga" son temporales porque las unidades productivas están pensadas para estar trabajando constantemente.
   VAR_INPUT
      start : Bool;
      emer : Bool;
      rearme : Bool;
      cong : Bool;
      dc : Bool;
      fin_p : Bool;
      home : Bool;
      tiempo_max : S5Time;
      temp_max : Timer;
   END_VAR
   VAR_OUTPUT
      cargar : Bool;
      descargar : Bool;
      bit_standby : Bool;
      bit_ocupacion : Bool;
      bit_error_tiempo_carga : Bool;
      bit_error_tiempo_descarga : Bool;
      bit_error_config_carga : Bool;
      bit_error_config_descarga : Bool;
      bit_emer : Bool;
   END_VAR
   VAR
      bit_trabajo : Bool;
      x_carga : Bool;
      x_descarga : Bool;
      x_standby : Bool;
      x_error_tiempo_carga : Bool;
      x_error_tiempo_descarga : Bool;
      x_error_config_carga : Bool;
      x_error_config_descarga : Bool;
      x_espera_home_carga : Bool;
      x_espera_home_descarga : Bool;
      x_emer : Bool;
      SFC_Programa_Carga : "SFC_Programa";
      SFC1_Programa_Descarga : "SFC_Programa";
   END_VAR
   VAR_TEMP
      bit_fin_carga : Bool;
      bit_fin_descarga : Bool;
   END_VAR
BEGIN

REGION Network 1: Plantilla de desconexion - Error asíncrono
   // Si se está en un estado de error síncrono no se entra en emergencia.
         O     #x_standby;
         O     #x_carga;
         O     #x_descarga;
         A     #emer;
         S     #x_emer;
         R     #x_standby;
         R     #x_carga;
         R     #x_descarga;

         JCN   _emer;

         CALL  #SFC_Programa_Carga
         ( sensor1          := ,
           sensor2          := ,
           reset            := true,
           tiempo_error     := ,
           temp_error       := #temp_max,
           bit_fin          := #bit_fin_carga,
           bit_error_tiempo := ,
           bit_error_config := ,
           bit_ocupacion    := #bit_ocupacion,
           actuador1        := #cargar
         );

         CALL  #SFC1_Programa_Descarga
         ( sensor1          := ,
           sensor2          := ,
           reset            := true,
           tiempo_error     := ,
           temp_error       := #temp_max,
           bit_fin          := #bit_fin_descarga,
           bit_error_tiempo := ,
           bit_error_config := ,
           bit_ocupacion    := #bit_ocupacion,
           actuador1        := #descargar
         );

   _emer:NOP   0;

         O     #x_standby;
         O     #x_carga;
         O     #x_descarga;
         A     #emer;
         BEC;
END_REGION

REGION Network 2: Plantilla de desconexión - STOP
   // Desconexión de la unidad productiva. 
   // Reinicia todos los parámetros para futuras conexiones.
   // Llamada a las maniobras usando la entrada asíncrona para indicar su pausa.
   // Después de la caja de código se especifica la instrucción “UN #start”, que coincide con la instrucción con la que se activó la plantilla. Esto es porque después de la caja, la RLO = 1 y /ER = 0. Por lo tanto, si la plantilla no se ejecuta, tras saltar la caja de código la RLO = 1 cuando debería ser 0 (UN #start no se cumple).
         AN    #start;
         R     #bit_trabajo;
         R     #bit_emer;
         R     #bit_error_config_carga;
         R     #bit_error_config_descarga;
         R     #bit_error_tiempo_carga;
         R     #bit_error_tiempo_descarga;
         R     #bit_standby;
         R     #bit_ocupacion;
         R     #temp_max;
         FR    #temp_max;

         JCN   stop;

         CALL  #SFC_Programa_Carga
         ( sensor1          := ,
           sensor2          := ,
           reset            := true,
           tiempo_error     := ,
           temp_error       := ,
           bit_fin          := ,
           bit_error_tiempo := ,
           bit_error_config := ,
           bit_ocupacion    := ,
           actuador1        := #cargar
         );

         CALL  #SFC1_Programa_Descarga
         ( sensor1          := ,
           sensor2          := ,
           reset            := true,
           tiempo_error     := ,
           temp_error       := ,
           bit_fin          := ,
           bit_error_tiempo := ,
           bit_error_config := ,
           bit_ocupacion    := ,
           actuador1        := #descargar
         );

   stop: NOP   0;

         AN    #start;
         BEC;
END_REGION

REGION Network 3: Plantilla de conexión
   // Conexión de la unidad productiva.
         A     #start;
         FP    #bit_trabajo;
         S     #x_standby;
         R     #x_carga;
         R     #x_descarga;
         R     #x_emer;
         R     #x_error_config_carga;
         R     #x_error_config_descarga;
         R     #x_error_tiempo_carga;
         R     #x_error_tiempo_descarga;
         R     #x_espera_home_carga;
         R     #x_espera_home_descarga;
END_REGION

REGION Network 4: Plantilla de congelación
   // Congela la unidad productiva: habilita los componentes y resetea los actuadores (llamadas a maniobras).
   // Se repite el estimulo de activación de la plantilla antes de la instrucción "BEB" para asegurar la salida del bloque.
         A     #cong;

         JCN   _cong;

         R     #temp_max;  //Habilitación de componentes
         FR    #temp_max;

         CALL  #SFC_Programa_Carga
         ( sensor1          := ,
           sensor2          := ,
           reset            := TRUE,
           tiempo_error     := ,
           temp_error       := ,
           bit_fin          := ,
           bit_error_tiempo := ,
           bit_error_config := ,
           bit_ocupacion    := ,
           actuador1        := #cargar
         );

         CALL  #SFC1_Programa_Descarga
         ( sensor1          := ,
           sensor2          := ,
           reset            := TRUE,
           tiempo_error     := ,
           temp_error       := ,
           bit_fin          := ,
           bit_error_tiempo := ,
           bit_error_config := ,
           bit_ocupacion    := ,
           actuador1        := #descargar
         );

   _cong:NOP   0;

         A     #cong;  //Repetición del estímulo de activación
         BEC;
END_REGION

REGION Network 5: Salida del estado de emergencia
   // Rearme. Necesaria la señal home (el robot tiene que estar en posición fetal para
   // estar en el estado de standby).
         A     #x_emer;
         AN    #emer;
         A     #rearme;
         S     #x_standby;
         R     #x_emer;
END_REGION

REGION Network 6: Rearme errores síncronos
   // Se considera la posibilidad de rearme tras errores síncronos.
         O     #x_error_config_carga;
         O     #x_error_config_descarga;
         O     #x_error_tiempo_carga;
         O     #x_error_tiempo_descarga;
         A     #rearme;
         S     #x_standby;
         R     #x_error_config_carga;
         R     #x_error_config_descarga;
         R     #x_error_tiempo_carga;
         R     #x_error_tiempo_descarga;
END_REGION

